LIN {X 0,Y 426.471,Z 695.747,A -85,B 0,C 180,E1 10312.845,E2 10312.845} C_VEL
LIN {X 0,Y 420.657,Z 731.018,A -85,B 0,C 180,E1 10315.887,E2 10315.887} C_VEL
LIN {X 0,Y 414.924,Z 763.236,A -85,B 0,C 180,E1 10319.677,E2 10319.677} C_VEL
LIN {X 0,Y 409.909,Z 791.343,A -85,B 0,C 180,E1 10324.089,E2 10324.089} C_VEL
LIN {X 0,Y 406.178,Z 814.952,A -85,B 0,C 180,E1 10329.05,E2 10329.05} C_VEL
LIN {X 0,Y 403.918,Z 833.153,A -85,B 0,C 180,E1 10334.286,E2 10334.286} C_VEL
LIN {X 0,Y 403.628,Z 836.352,A -85,B 0,C 180,E1 10335.425,E2 10335.425} C_VEL
LIN {X 0,Y 400.755,Z 840.636,A -85,B 0,C 180,E1 10337.153,E2 10337.153} C_VEL
LIN {X 0,Y 395.126,Z 845.824,A -85,B 0,C 180,E1 10339.793,E2 10339.793} C_VEL
LIN {X 0,Y 395.001,Z 846.38,A -85,B 0,C 180,E1 10340.101,E2 10340.101} C_VEL
LIN {X 0,Y 394.597,Z 853.166,A -85,B 0,C 180,E1 10345.615,E2 10345.615} C_VEL
LIN {X 0,Y 394.715,Z 854.908,A -85,B 0,C 180,E1 10350.002,E2 10350.002} C_VEL
LIN {X 0,Y 394.613,Z 853.222,A -85,B 0,C 180,E1 10354.388,E2 10354.388} C_VEL
LIN {X 0,Y 394.945,Z 846.511,A -85,B 0,C 180,E1 10359.902,E2 10359.902} C_VEL
LIN {X 0,Y 395.944,Z 834.241,A -85,B 0,C 180,E1 10365.475,E2 10365.475} C_VEL
LIN {X 0,Y 398.38,Z 815.704,A -85,B 0,C 180,E1 10371.093,E2 10371.093} C_VEL
LIN {X 0,Y 402.285,Z 792.827,A -85,B 0,C 180,E1 10376.109,E2 10376.109} C_VEL
LIN {X 0,Y 407.51,Z 765.346,A -85,B 0,C 180,E1 10380.61,E2 10380.61} C_VEL
LIN {X 0,Y 413.404,Z 734.349,A -85,B 0,C 180,E1 10384.414,E2 10384.414} C_VEL
LIN {X 0,Y 419.63,Z 699.188,A -85,B 0,C 180,E1 10387.577,E2 10387.577} C_VEL
LIN {X 0,Y 424.895,Z 663.712,A -85,B 0,C 180,E1 10389.841,E2 10389.841} C_VEL
LIN {X 0,Y 429.031,Z 626.267,A -85,B 0,C 180,E1 10391.417,E2 10391.417} C_VEL
LIN {X 0,Y 428.573,Z 619.383,A -85,B 0,C 180,E1 10391.743,E2 10391.743} C_VEL
LIN {X 0,Y 412.157,Z 584.483,A -85,B 0,C 180,E1 10394.597,E2 10394.597} C_VEL
LIN {X 0,Y 393.303,Z 551.113,A -85,B 0,C 180,E1 10397.831,E2 10397.831} C_VEL
LIN {X 0,Y 393.107,Z 549.53,A -85,B 0,C 180,E1 10397.988,E2 10397.988} C_VEL
LIN {X 0,Y 393.066,Z 549.53,A -85,B 0,C 180,E1 10404.827,E2 10404.827} C_VEL
LIN {X 0,Y 393.133,Z 549.53,A -85,B 0,C 180,E1 10411.99,E2 10411.99} C_VEL
LIN {X 0,Y 393.428,Z 549.53,A -85,B 0,C 180,E1 10417.432,E2 10417.432} C_VEL
LIN {X 0,Y 393.65,Z 549.53,A -85,B 0,C 180,E1 10424.419,E2 10424.419} C_VEL
LIN {X 0,Y 393.977,Z 549.53,A -85,B 0,C 180,E1 10431.171,E2 10431.171} C_VEL
LIN {X 0,Y 394.49,Z 549.53,A -85,B 0,C 180,E1 10437.79,E2 10437.79} C_VEL
LIN {X 0,Y 394.273,Z 549.53,A -85,B 0,C 180,E1 10444.371,E2 10444.371} C_VEL
LIN {X 0,Y 393.966,Z 549.53,A -85,B 0,C 180,E1 10451.02,E2 10451.02} C_VEL
LIN {X 0,Y 393.651,Z 549.53,A -85,B 0,C 180,E1 10457.835,E2 10457.835} C_VEL
LIN {X 0,Y 393.41,Z 549.53,A -85,B 0,C 180,E1 10464.93,E2 10464.93} C_VEL
LIN {X 0,Y 393.257,Z 549.53,A -85,B 0,C 180,E1 10472.464,E2 10472.464} C_VEL
LIN {X 0,Y 393.138,Z 549.53,A -85,B 0,C 180,E1 10479.852,E2 10479.852} C_VEL
LIN {X 0,Y 393.035,Z 549.53,A -85,B 0,C 180,E1 10486.802,E2 10486.802} C_VEL
LIN {X 0,Y 393.151,Z 549.53,A -85,B 0,C 180,E1 10493.661,E2 10493.661} C_VEL
LIN {X 0,Y 393.294,Z 549.53,A -85,B 0,C 180,E1 10500.078,E2 10500.078} C_VEL
LIN {X 0,Y 393.473,Z 549.53,A -85,B 0,C 180,E1 10507.447,E2 10507.447} C_VEL
LIN {X 0,Y 393.748,Z 549.858,A -85,B 0,C 180,E1 10514.366,E2 10514.366} C_VEL
LIN {X 0,Y 398.982,Z 560.257,A -85,B 0,C 180,E1 10515.316,E2 10515.316} C_VEL
LIN {X 0,Y 415.159,Z 593.265,A -85,B 0,C 180,E1 10518.486,E2 10518.486} C_VEL
LIN {X 0,Y 422.389,Z 615.31,A -85,B 0,C 180,E1 10520.492,E2 10520.492} C_VEL
LIN {X 0,Y 417.734,Z 650.048,A -85,B 0,C 180,E1 10522.702,E2 10522.702} C_VEL
LIN {X 0,Y 412.529,Z 681.161,A -85,B 0,C 180,E1 10525.54,E2 10525.54} C_VEL
LIN {X 0,Y 406.889,Z 710.862,A -85,B 0,C 180,E1 10529.292,E2 10529.292} C_VEL
LIN {X 0,Y 401.898,Z 736.31,A -85,B 0,C 180,E1 10533.766,E2 10533.766} C_VEL
LIN {X 0,Y 398.293,Z 756.361,A -85,B 0,C 180,E1 10538.715,E2 10538.715} C_VEL
LIN {X 0,Y 396.006,Z 771.387,A -85,B 0,C 180,E1 10544.145,E2 10544.145} C_VEL
LIN {X 0,Y 395.061,Z 779.568,A -85,B 0,C 180,E1 10548.944,E2 10548.944} C_VEL
LIN {X 0,Y 394.329,Z 783.387,A -85,B 0,C 180,E1 10553.38,E2 10553.38} C_VEL
LIN {X 0,Y 394.392,Z 783.535,A -85,B 0,C 180,E1 10558.419,E2 10558.419} C_VEL
LIN {X 0,Y 395.372,Z 778.667,A -85,B 0,C 180,E1 10563.847,E2 10563.847} C_VEL
LIN {X 0,Y 396.658,Z 768.466,A -85,B 0,C 180,E1 10569.268,E2 10569.268} C_VEL
LIN {X 0,Y 399.169,Z 752.985,A -85,B 0,C 180,E1 10574.422,E2 10574.422} C_VEL
LIN {X 0,Y 403.09,Z 732.77,A -85,B 0,C 180,E1 10579.115,E2 10579.115} C_VEL
LIN {X 0,Y 408.186,Z 708.039,A -85,B 0,C 180,E1 10583.279,E2 10583.279} C_VEL
LIN {X 0,Y 413.987,Z 678.023,A -85,B 0,C 180,E1 10586.965,E2 10586.965} C_VEL
LIN {X 0,Y 419.505,Z 645.504,A -85,B 0,C 180,E1 10589.789,E2 10589.789} C_VEL
LIN {X 0,Y 423.419,Z 614.726,A -85,B 0,C 180,E1 10591.704,E2 10591.704} C_VEL
LIN {X 0,Y 410.683,Z 582.196,A -85,B 0,C 180,E1 10594.957,E2 10594.957} C_VEL
LIN {X 0,Y 395.046,Z 554.114,A -85,B 0,C 180,E1 10598.086,E2 10598.086} C_VEL
LIN {X 0,Y 393.557,Z 549.53,A -85,B 0,C 180,E1 10598.516,E2 10598.516} C_VEL
LIN {X 0,Y 393.66,Z 549.53,A -85,B 0,C 180,E1 10604.458,E2 10604.458} C_VEL
LIN {X 0,Y 393.997,Z 549.53,A -85,B 0,C 180,E1 10611.208,E2 10611.208} C_VEL
LIN {X 0,Y 394.47,Z 549.53,A -85,B 0,C 180,E1 10617.826,E2 10617.826} C_VEL
LIN {X 0,Y 394.267,Z 549.53,A -85,B 0,C 180,E1 10624.407,E2 10624.407} C_VEL
LIN {X 0,Y 393.97,Z 549.53,A -85,B 0,C 180,E1 10631.057,E2 10631.057} C_VEL
LIN {X 0,Y 393.667,Z 549.53,A -85,B 0,C 180,E1 10637.873,E2 10637.873} C_VEL
LIN {X 0,Y 393.385,Z 549.53,A -85,B 0,C 180,E1 10644.972,E2 10644.972} C_VEL
LIN {X 0,Y 393.268,Z 549.53,A -85,B 0,C 180,E1 10652.506,E2 10652.506} C_VEL
LIN {X 0,Y 393.117,Z 549.53,A -85,B 0,C 180,E1 10659.853,E2 10659.853} C_VEL
LIN {X 0,Y 393.019,Z 549.552,A -85,B 0,C 180,E1 10661.786,E2 10661.786} C_VEL
LIN {X 0,Y 395.349,Z 555.078,A -85,B 0,C 180,E1 10662.289,E2 10662.289} C_VEL
LIN {X 0,Y 414.303,Z 587.868,A -85,B 0,C 180,E1 10665.71,E2 10665.71} C_VEL
LIN {X 0,Y 429.06,Z 620.928,A -85,B 0,C 180,E1 10668.451,E2 10668.451} C_VEL
LIN {X 0,Y 424.831,Z 660.824,A -85,B 0,C 180,E1 10670.072,E2 10670.072} C_VEL
LIN {X 0,Y 419.322,Z 698.722,A -85,B 0,C 180,E1 10672.477,E2 10672.477} C_VEL
LIN {X 0,Y 413.275,Z 733.396,A -85,B 0,C 180,E1 10675.601,E2 10675.601} C_VEL
LIN {X 0,Y 407.388,Z 764.437,A -85,B 0,C 180,E1 10679.384,E2 10679.384} C_VEL
LIN {X 0,Y 402.203,Z 792.195,A -85,B 0,C 180,E1 10683.894,E2 10683.894} C_VEL
LIN {X 0,Y 398.349,Z 815.265,A -85,B 0,C 180,E1 10688.909,E2 10688.909} C_VEL
LIN {X 0,Y 395.954,Z 833.988,A -85,B 0,C 180,E1 10694.529,E2 10694.529} C_VEL
LIN {X 0,Y 395.001,Z 846.38,A -85,B 0,C 180,E1 10700.101,E2 10700.101} C_VEL
LIN {X 0,Y 392.28,Z 849.129,A -85,B 0,C 180,E1 10701.929,E2 10701.929} C_VEL
LIN {X 0,Y 386.796,Z 851.796,A -85,B 0,C 180,E1 10704.721,E2 10704.721} C_VEL
LIN {X 0,Y 386.707,Z 852.052,A -85,B 0,C 180,E1 10705.046,E2 10705.046} C_VEL
LIN {X 0,Y 386.852,Z 854.204,A -85,B 0,C 180,E1 10710.002,E2 10710.002} C_VEL
LIN {X 0,Y 386.746,Z 852.519,A -85,B 0,C 180,E1 10714.477,E2 10714.477} C_VEL
LIN {X 0,Y 387.089,Z 845.8,A -85,B 0,C 180,E1 10720.105,E2 10720.105} C_VEL
LIN {X 0,Y 388.13,Z 833.511,A -85,B 0,C 180,E1 10725.794,E2 10725.794} C_VEL
LIN {X 0,Y 390.582,Z 815.874,A -85,B 0,C 180,E1 10731.288,E2 10731.288} C_VEL
LIN {X 0,Y 394.703,Z 793.039,A -85,B 0,C 180,E1 10736.444,E2 10736.444} C_VEL
LIN {X 0,Y 400.02,Z 766.445,A -85,B 0,C 180,E1 10740.931,E2 10740.931} C_VEL
LIN {X 0,Y 406.373,Z 734.587,A -85,B 0,C 180,E1 10744.942,E2 10744.942} C_VEL
LIN {X 0,Y 412.893,Z 699.726,A -85,B 0,C 180,E1 10748.14,E2 10748.14} C_VEL
LIN {X 0,Y 418.485,Z 663.769,A -85,B 0,C 180,E1 10750.473,E2 10750.473} C_VEL
LIN {X 0,Y 422.776,Z 626.655,A -85,B 0,C 180,E1 10752.06,E2 10752.06} C_VEL
LIN {X 0,Y 421.658,Z 620.596,A -85,B 0,C 180,E1 10752.433,E2 10752.433} C_VEL
LIN {X 0,Y 405.945,Z 587.248,A -85,B 0,C 180,E1 10755.297,E2 10755.297} C_VEL
LIN {X 0,Y 386.357,Z 553.583,A -85,B 0,C 180,E1 10758.759,E2 10758.759} C_VEL
LIN {X 0,Y 385.217,Z 549.53,A -85,B 0,C 180,E1 10759.111,E2 10759.111} C_VEL
LIN {X 0,Y 385.118,Z 549.53,A -85,B 0,C 180,E1 10766.718,E2 10766.718} C_VEL
LIN {X 0,Y 385.314,Z 549.53,A -85,B 0,C 180,E1 10774.261,E2 10774.261} C_VEL
LIN {X 0,Y 385.665,Z 549.53,A -85,B 0,C 180,E1 10779.899,E2 10779.899} C_VEL
LIN {X 0,Y 385.782,Z 549.53,A -85,B 0,C 180,E1 10786.41,E2 10786.41} C_VEL
LIN {X 0,Y 386.241,Z 549.53,A -85,B 0,C 180,E1 10793.252,E2 10793.252} C_VEL
LIN {X 0,Y 386.542,Z 549.53,A -85,B 0,C 180,E1 10799.981,E2 10799.981} C_VEL
LIN {X 0,Y 386.242,Z 549.53,A -85,B 0,C 180,E1 10806.711,E2 10806.711} C_VEL
LIN {X 0,Y 385.971,Z 549.53,A -85,B 0,C 180,E1 10813.544,E2 10813.544} C_VEL
LIN {X 0,Y 385.622,Z 549.53,A -85,B 0,C 180,E1 10820.596,E2 10820.596} C_VEL
LIN {X 0,Y 385.391,Z 549.53,A -85,B 0,C 180,E1 10827.997,E2 10827.997} C_VEL
LIN {X 0,Y 385.257,Z 549.53,A -85,B 0,C 180,E1 10835.949,E2 10835.949} C_VEL
LIN {X 0,Y 385.08,Z 549.53,A -85,B 0,C 180,E1 10841.877,E2 10841.877} C_VEL
LIN {X 0,Y 385.068,Z 549.53,A -85,B 0,C 180,E1 10848.223,E2 10848.223} C_VEL
LIN {X 0,Y 385.242,Z 549.53,A -85,B 0,C 180,E1 10854.014,E2 10854.014} C_VEL
LIN {X 0,Y 385.337,Z 549.53,A -85,B 0,C 180,E1 10859.43,E2 10859.43} C_VEL
LIN {X 0,Y 385.58,Z 549.53,A -85,B 0,C 180,E1 10866.959,E2 10866.959} C_VEL
LIN {X 0,Y 385.772,Z 549.53,A -85,B 0,C 180,E1 10873.251,E2 10873.251} C_VEL
LIN {X 0,Y 388.253,Z 555.254,A -85,B 0,C 180,E1 10873.76,E2 10873.76} C_VEL
LIN {X 0,Y 405.744,Z 588.831,A -85,B 0,C 180,E1 10877.194,E2 10877.194} C_VEL
LIN {X 0,Y 415.978,Z 616.303,A -85,B 0,C 180,E1 10879.879,E2 10879.879} C_VEL
LIN {X 0,Y 411.293,Z 649.927,A -85,B 0,C 180,E1 10882.038,E2 10882.038} C_VEL
LIN {X 0,Y 405.76,Z 681.449,A -85,B 0,C 180,E1 10884.931,E2 10884.931} C_VEL
LIN {X 0,Y 400.146,Z 709.999,A -85,B 0,C 180,E1 10888.562,E2 10888.562} C_VEL
LIN {X 0,Y 394.861,Z 735.482,A -85,B 0,C 180,E1 10893.01,E2 10893.01} C_VEL
LIN {X 0,Y 391.051,Z 754.99,A -85,B 0,C 180,E1 10897.76,E2 10897.76} C_VEL
LIN {X 0,Y 388.554,Z 769.773,A -85,B 0,C 180,E1 10902.902,E2 10902.902} C_VEL
LIN {X 0,Y 387.354,Z 779.383,A -85,B 0,C 180,E1 10908.157,E2 10908.157} C_VEL
LIN {X 0,Y 386.51,Z 783.925,A -85,B 0,C 180,E1 10912.979,E2 10912.979} C_VEL
LIN {X 0,Y 386.471,Z 784.476,A -85,B 0,C 180,E1 10917.938,E2 10917.938} C_VEL
LIN {X 0,Y 387.377,Z 780.657,A -85,B 0,C 180,E1 10923.048,E2 10923.048} C_VEL
LIN {X 0,Y 388.494,Z 771.732,A -85,B 0,C 180,E1 10928.422,E2 10928.422} C_VEL
LIN {X 0,Y 390.929,Z 757.617,A -85,B 0,C 180,E1 10933.652,E2 10933.652} C_VEL
LIN {X 0,Y 394.939,Z 737.673,A -85,B 0,C 180,E1 10938.728,E2 10938.728} C_VEL
LIN {X 0,Y 400.489,Z 712.216,A -85,B 0,C 180,E1 10943.311,E2 10943.311} C_VEL
LIN {X 0,Y 406.474,Z 683.127,A -85,B 0,C 180,E1 10947.082,E2 10947.082} C_VEL
LIN {X 0,Y 412.498,Z 650.226,A -85,B 0,C 180,E1 10950.129,E2 10950.129} C_VEL
LIN {X 0,Y 416.669,Z 616.289,A -85,B 0,C 180,E1 10952.38,E2 10952.38} C_VEL
LIN {X 0,Y 403.829,Z 583.58,A -85,B 0,C 180,E1 10955.816,E2 10955.816} C_VEL
LIN {X 0,Y 388.017,Z 555.131,A -85,B 0,C 180,E1 10959.166,E2 10959.166} C_VEL
LIN {X 0,Y 385.726,Z 549.53,A -85,B 0,C 180,E1 10959.865,E2 10959.865} C_VEL
LIN {X 0,Y 385.803,Z 549.53,A -85,B 0,C 180,E1 10966.45,E2 10966.45} C_VEL
LIN {X 0,Y 386.278,Z 549.53,A -85,B 0,C 180,E1 10973.29,E2 10973.29} C_VEL
LIN {X 0,Y 386.548,Z 549.53,A -85,B 0,C 180,E1 10980.019,E2 10980.019} C_VEL
LIN {X 0,Y 386.244,Z 549.53,A -85,B 0,C 180,E1 10986.748,E2 10986.748} C_VEL
LIN {X 0,Y 385.991,Z 549.53,A -85,B 0,C 180,E1 10993.582,E2 10993.582} C_VEL
LIN {X 0,Y 385.615,Z 549.53,A -85,B 0,C 180,E1 11000.636,E2 11000.636} C_VEL
LIN {X 0,Y 385.387,Z 549.53,A -85,B 0,C 180,E1 11008.04,E2 11008.04} C_VEL
LIN {X 0,Y 385.233,Z 549.53,A -85,B 0,C 180,E1 11014.657,E2 11014.657} C_VEL
LIN {X 0,Y 385.198,Z 549.884,A -85,B 0,C 180,E1 11020.518,E2 11020.518} C_VEL
LIN {X 0,Y 387.642,Z 555.268,A -85,B 0,C 180,E1 11021.073,E2 11021.073} C_VEL
LIN {X 0,Y 406.583,Z 587.415,A -85,B 0,C 180,E1 11024.695,E2 11024.695} C_VEL
LIN {X 0,Y 421.438,Z 620.064,A -85,B 0,C 180,E1 11027.575,E2 11027.575} C_VEL
LIN {X 0,Y 422.509,Z 626.284,A -85,B 0,C 180,E1 11027.955,E2 11027.955} C_VEL
LIN {X 0,Y 417.796,Z 666.137,A -85,B 0,C 180,E1 11029.705,E2 11029.705} C_VEL
LIN {X 0,Y 411.485,Z 705.521,A -85,B 0,C 180,E1 11032.405,E2 11032.405} C_VEL
LIN {X 0,Y 404.886,Z 740.387,A -85,B 0,C 180,E1 11035.816,E2 11035.816} C_VEL
LIN {X 0,Y 398.767,Z 771.137,A -85,B 0,C 180,E1 11039.909,E2 11039.909} C_VEL
LIN {X 0,Y 393.725,Z 797.105,A -85,B 0,C 180,E1 11044.51,E2 11044.51} C_VEL
LIN {X 0,Y 389.994,Z 819.77,A -85,B 0,C 180,E1 11049.917,E2 11049.917} C_VEL
LIN {X 0,Y 387.878,Z 836.124,A -85,B 0,C 180,E1 11055.354,E2 11055.354} C_VEL
LIN {X 0,Y 386.98,Z 847.395,A -85,B 0,C 180,E1 11061.028,E2 11061.028} C_VEL
LIN {X 0,Y 386.707,Z 852.052,A -85,B 0,C 180,E1 11065.046,E2 11065.046} C_VEL
LIN {X 0,Y 384.331,Z 853.217,A -85,B 0,C 180,E1 11066.952,E2 11066.952} C_VEL
LIN {X 0,Y 378.98,Z 853.469,A -85,B 0,C 180,E1 11070.169,E2 11070.169} C_VEL
LIN {X 0,Y 378.856,Z 851.309,A -85,B 0,C 180,E1 11075.212,E2 11075.212} C_VEL
LIN {X 0,Y 379.22,Z 845.088,A -85,B 0,C 180,E1 11080.317,E2 11080.317} C_VEL
LIN {X 0,Y 380.334,Z 832.776,A -85,B 0,C 180,E1 11086.127,E2 11086.127} C_VEL
LIN {X 0,Y 382.893,Z 815.414,A -85,B 0,C 180,E1 11091.654,E2 11091.654} C_VEL
LIN {X 0,Y 387.461,Z 791.705,A -85,B 0,C 180,E1 11097.086,E2 11097.086} C_VEL
LIN {X 0,Y 393.329,Z 763.563,A -85,B 0,C 180,E1 11101.84,E2 11101.84} C_VEL
LIN {X 0,Y 399.84,Z 732.637,A -85,B 0,C 180,E1 11105.722,E2 11105.722} C_VEL
LIN {X 0,Y 406.572,Z 698.065,A -85,B 0,C 180,E1 11108.888,E2 11108.888} C_VEL
LIN {X 0,Y 412.308,Z 662.252,A -85,B 0,C 180,E1 11111.209,E2 11111.209} C_VEL
LIN {X 0,Y 416.143,Z 625.507,A -85,B 0,C 180,E1 11112.836,E2 11112.836} C_VEL
LIN {X 0,Y 400.463,Z 591.124,A -85,B 0,C 180,E1 11115.903,E2 11115.903} C_VEL
LIN {X 0,Y 379.231,Z 554.747,A -85,B 0,C 180,E1 11119.79,E2 11119.79} C_VEL
LIN {X 0,Y 377.267,Z 549.53,A -85,B 0,C 180,E1 11120.323,E2 11120.323} C_VEL
LIN {X 0,Y 377.174,Z 549.53,A -85,B 0,C 180,E1 11127.162,E2 11127.162} C_VEL
LIN {X 0,Y 377.369,Z 549.53,A -85,B 0,C 180,E1 11133.89,E2 11133.89} C_VEL
LIN {X 0,Y 377.629,Z 549.53,A -85,B 0,C 180,E1 11138.907,E2 11138.907} C_VEL
LIN {X 0,Y 377.84,Z 549.53,A -85,B 0,C 180,E1 11146.119,E2 11146.119} C_VEL
LIN {X 0,Y 378.321,Z 549.53,A -85,B 0,C 180,E1 11153.11,E2 11153.11} C_VEL
LIN {X 0,Y 378.64,Z 549.53,A -85,B 0,C 180,E1 11159.981,E2 11159.981} C_VEL
LIN {X 0,Y 378.323,Z 549.53,A -85,B 0,C 180,E1 11166.852,E2 11166.852} C_VEL
LIN {X 0,Y 378.018,Z 549.53,A -85,B 0,C 180,E1 11173.835,E2 11173.835} C_VEL
LIN {X 0,Y 377.654,Z 549.53,A -85,B 0,C 180,E1 11181.051,E2 11181.051} C_VEL
LIN {X 0,Y 377.412,Z 549.53,A -85,B 0,C 180,E1 11188.643,E2 11188.643} C_VEL
LIN {X 0,Y 377.316,Z 549.53,A -85,B 0,C 180,E1 11194.017,E2 11194.017} C_VEL
LIN {X 0,Y 377.128,Z 549.53,A -85,B 0,C 180,E1 11200.511,E2 11200.511} C_VEL
LIN {X 0,Y 377.055,Z 549.53,A -85,B 0,C 180,E1 11207.126,E2 11207.126} C_VEL
LIN {X 0,Y 377.278,Z 549.53,A -85,B 0,C 180,E1 11213.131,E2 11213.131} C_VEL
LIN {X 0,Y 377.315,Z 549.53,A -85,B 0,C 180,E1 11218.671,E2 11218.671} C_VEL
LIN {X 0,Y 377.485,Z 549.53,A -85,B 0,C 180,E1 11223.911,E2 11223.911} C_VEL
LIN {X 0,Y 377.655,Z 549.53,A -85,B 0,C 180,E1 11228.921,E2 11228.921} C_VEL
LIN {X 0,Y 377.839,Z 550.299,A -85,B 0,C 180,E1 11232.134,E2 11232.134} C_VEL
LIN {X 0,Y 386.756,Z 566.255,A -85,B 0,C 180,E1 11233.872,E2 11233.872} C_VEL
LIN {X 0,Y 402.213,Z 598.37,A -85,B 0,C 180,E1 11237.249,E2 11237.249} C_VEL
LIN {X 0,Y 409.274,Z 619.687,A -85,B 0,C 180,E1 11239.375,E2 11239.375} C_VEL
LIN {X 0,Y 404.372,Z 652.868,A -85,B 0,C 180,E1 11241.596,E2 11241.596} C_VEL
LIN {X 0,Y 398.419,Z 685.269,A -85,B 0,C 180,E1 11244.701,E2 11244.701} C_VEL
LIN {X 0,Y 392.241,Z 714.458,A -85,B 0,C 180,E1 11248.61,E2 11248.61} C_VEL
LIN {X 0,Y 387.03,Z 738.331,A -85,B 0,C 180,E1 11253.032,E2 11253.032} C_VEL
LIN {X 0,Y 383.147,Z 757.412,A -85,B 0,C 180,E1 11257.922,E2 11257.922} C_VEL
LIN {X 0,Y 380.662,Z 771.669,A -85,B 0,C 180,E1 11263.174,E2 11263.174} C_VEL
LIN {X 0,Y 379.412,Z 780.815,A -85,B 0,C 180,E1 11268.551,E2 11268.551} C_VEL
LIN {X 0,Y 378.56,Z 784.947,A -85,B 0,C 180,E1 11273.612,E2 11273.612} C_VEL
LIN {X 0,Y 378.668,Z 784.848,A -85,B 0,C 180,E1 11278.816,E2 11278.816} C_VEL
LIN {X 0,Y 379.698,Z 780.606,A -85,B 0,C 180,E1 11283.805,E2 11283.805} C_VEL
LIN {X 0,Y 381.021,Z 771.083,A -85,B 0,C 180,E1 11289.319,E2 11289.319} C_VEL
LIN {X 0,Y 383.821,Z 756.168,A -85,B 0,C 180,E1 11294.707,E2 11294.707} C_VEL
LIN {X 0,Y 388.411,Z 735.173,A -85,B 0,C 180,E1 11299.888,E2 11299.888} C_VEL
LIN {X 0,Y 394.245,Z 709.826,A -85,B 0,C 180,E1 11304.335,E2 11304.335} C_VEL
LIN {X 0,Y 400.47,Z 680.842,A -85,B 0,C 180,E1 11308.032,E2 11308.032} C_VEL
LIN {X 0,Y 406.786,Z 647.048,A -85,B 0,C 180,E1 11311.08,E2 11311.08} C_VEL
LIN {X 0,Y 410.49,Z 619.762,A -85,B 0,C 180,E1 11312.878,E2 11312.878} C_VEL
LIN {X 0,Y 398.576,Z 588.31,A -85,B 0,C 180,E1 11316.32,E2 11316.32} C_VEL
LIN {X 0,Y 383.84,Z 561.006,A -85,B 0,C 180,E1 11319.68,E2 11319.68} C_VEL
LIN {X 0,Y 377.85,Z 550.7,A -85,B 0,C 180,E1 11321.051,E2 11321.051} C_VEL
LIN {X 0,Y 377.75,Z 549.53,A -85,B 0,C 180,E1 11321.387,E2 11321.387} C_VEL
LIN {X 0,Y 377.972,Z 549.53,A -85,B 0,C 180,E1 11328.507,E2 11328.507} C_VEL
LIN {X 0,Y 378.437,Z 549.53,A -85,B 0,C 180,E1 11335.446,E2 11335.446} C_VEL
LIN {X 0,Y 378.522,Z 549.53,A -85,B 0,C 180,E1 11342.303,E2 11342.303} C_VEL
LIN {X 0,Y 378.167,Z 549.53,A -85,B 0,C 180,E1 11349.202,E2 11349.202} C_VEL
LIN {X 0,Y 377.888,Z 549.53,A -85,B 0,C 180,E1 11356.248,E2 11356.248} C_VEL
LIN {X 0,Y 377.554,Z 549.53,A -85,B 0,C 180,E1 11363.573,E2 11363.573} C_VEL
LIN {X 0,Y 377.416,Z 549.53,A -85,B 0,C 180,E1 11368.686,E2 11368.686} C_VEL
LIN {X 0,Y 377.316,Z 549.53,A -85,B 0,C 180,E1 11374.063,E2 11374.063} C_VEL
LIN {X 0,Y 377.31,Z 549.53,A -85,B 0,C 180,E1 11379.073,E2 11379.073} C_VEL
LIN {X 0,Y 379.801,Z 555.282,A -85,B 0,C 180,E1 11379.732,E2 11379.732} C_VEL
LIN {X 0,Y 398.809,Z 586.851,A -85,B 0,C 180,E1 11383.605,E2 11383.605} C_VEL
LIN {X 0,Y 413.991,Z 619.607,A -85,B 0,C 180,E1 11386.687,E2 11386.687} C_VEL
LIN {X 0,Y 416.364,Z 626.906,A -85,B 0,C 180,E1 11387.283,E2 11387.283} C_VEL
LIN {X 0,Y 411.311,Z 667.365,A -85,B 0,C 180,E1 11389.109,E2 11389.109} C_VEL
LIN {X 0,Y 404.88,Z 705.412,A -85,B 0,C 180,E1 11391.777,E2 11391.777} C_VEL
LIN {X 0,Y 398.055,Z 739.668,A -85,B 0,C 180,E1 11395.175,E2 11395.175} C_VEL
LIN {X 0,Y 391.625,Z 770.248,A -85,B 0,C 180,E1 11399.301,E2 11399.301} C_VEL
LIN {X 0,Y 386.151,Z 796.925,A -85,B 0,C 180,E1 11404.12,E2 11404.12} C_VEL
LIN {X 0,Y 382.272,Z 818.957,A -85,B 0,C 180,E1 11409.494,E2 11409.494} C_VEL
LIN {X 0,Y 380.047,Z 835.356,A -85,B 0,C 180,E1 11415.045,E2 11415.045} C_VEL
LIN {X 0,Y 379.112,Z 846.657,A -85,B 0,C 180,E1 11420.84,E2 11420.84} C_VEL
LIN {X 0,Y 378.849,Z 851.732,A -85,B 0,C 180,E1 11425.433,E2 11425.433} C_VEL
LIN {X 0,Y 378.98,Z 853.469,A -85,B 0,C 180,E1 11430.169,E2 11430.169} C_VEL
LIN {X 0,Y 376.344,Z 852.926,A -85,B 0,C 180,E1 11432.113,E2 11432.113} C_VEL
LIN {X 0,Y 370.977,Z 850.565,A -85,B 0,C 180,E1 11435.366,E2 11435.366} C_VEL
LIN {X 0,Y 371.342,Z 844.372,A -85,B 0,C 180,E1 11440.538,E2 11440.538} C_VEL
LIN {X 0,Y 372.556,Z 832.039,A -85,B 0,C 180,E1 11446.473,E2 11446.473} C_VEL
LIN {X 0,Y 375.503,Z 813.491,A -85,B 0,C 180,E1 11452.421,E2 11452.421} C_VEL
LIN {X 0,Y 380.244,Z 790.146,A -85,B 0,C 180,E1 11457.797,E2 11457.797} C_VEL
LIN {X 0,Y 386.345,Z 762.665,A -85,B 0,C 180,E1 11462.485,E2 11462.485} C_VEL
LIN {X 0,Y 393.184,Z 731.684,A -85,B 0,C 180,E1 11466.41,E2 11466.41} C_VEL
LIN {X 0,Y 400.235,Z 696.848,A -85,B 0,C 180,E1 11469.623,E2 11469.623} C_VEL
LIN {X 0,Y 406.363,Z 659.625,A -85,B 0,C 180,E1 11472.027,E2 11472.027} C_VEL
LIN {X 0,Y 409.851,Z 628.218,A -85,B 0,C 180,E1 11473.435,E2 11473.435} C_VEL
LIN {X 0,Y 394.517,Z 594.497,A -85,B 0,C 180,E1 11476.582,E2 11476.582} C_VEL
LIN {X 0,Y 374.605,Z 560.065,A -85,B 0,C 180,E1 11480.365,E2 11480.365} C_VEL
LIN {X 0,Y 369.429,Z 550.458,A -85,B 0,C 180,E1 11481.459,E2 11481.459} C_VEL
LIN {X 0,Y 369.384,Z 549.53,A -85,B 0,C 180,E1 11481.602,E2 11481.602} C_VEL
LIN {X 0,Y 369.249,Z 549.53,A -85,B 0,C 180,E1 11489.119,E2 11489.119} C_VEL
LIN {X 0,Y 369.527,Z 549.53,A -85,B 0,C 180,E1 11495.883,E2 11495.883} C_VEL
LIN {X 0,Y 369.849,Z 549.53,A -85,B 0,C 180,E1 11503.389,E2 11503.389} C_VEL
LIN {X 0,Y 370.162,Z 549.53,A -85,B 0,C 180,E1 11510.598,E2 11510.598} C_VEL
LIN {X 0,Y 370.762,Z 549.53,A -85,B 0,C 180,E1 11517.649,E2 11517.649} C_VEL
LIN {X 0,Y 370.539,Z 549.53,A -85,B 0,C 180,E1 11524.651,E2 11524.651} C_VEL
LIN {X 0,Y 370.163,Z 549.53,A -85,B 0,C 180,E1 11531.925,E2 11531.925} C_VEL
LIN {X 0,Y 369.799,Z 549.53,A -85,B 0,C 180,E1 11539.028,E2 11539.028} C_VEL
LIN {X 0,Y 369.499,Z 549.53,A -85,B 0,C 180,E1 11546.666,E2 11546.666} C_VEL
LIN {X 0,Y 369.425,Z 549.53,A -85,B 0,C 180,E1 11552.043,E2 11552.043} C_VEL
LIN {X 0,Y 369.227,Z 549.53,A -85,B 0,C 180,E1 11559.054,E2 11559.054} C_VEL
LIN {X 0,Y 369.141,Z 549.53,A -85,B 0,C 180,E1 11565.975,E2 11565.975} C_VEL
LIN {X 0,Y 369.254,Z 549.53,A -85,B 0,C 180,E1 11572.191,E2 11572.191} C_VEL
LIN {X 0,Y 369.397,Z 549.53,A -85,B 0,C 180,E1 11579.017,E2 11579.017} C_VEL
LIN {X 0,Y 369.611,Z 549.53,A -85,B 0,C 180,E1 11585.902,E2 11585.902} C_VEL
LIN {X 0,Y 369.773,Z 549.53,A -85,B 0,C 180,E1 11590.869,E2 11590.869} C_VEL
LIN {X 0,Y 372.261,Z 555.188,A -85,B 0,C 180,E1 11591.425,E2 11591.425} C_VEL
LIN {X 0,Y 389.181,Z 585.887,A -85,B 0,C 180,E1 11594.967,E2 11594.967} C_VEL
LIN {X 0,Y 401.619,Z 617.364,A -85,B 0,C 180,E1 11598.334,E2 11598.334} C_VEL
LIN {X 0,Y 402.526,Z 623.665,A -85,B 0,C 180,E1 11598.89,E2 11598.89} C_VEL
LIN {X 0,Y 397.073,Z 658.603,A -85,B 0,C 180,E1 11601.378,E2 11601.378} C_VEL
LIN {X 0,Y 390.749,Z 690.115,A -85,B 0,C 180,E1 11604.597,E2 11604.597} C_VEL
LIN {X 0,Y 384.479,Z 718.191,A -85,B 0,C 180,E1 11608.582,E2 11608.582} C_VEL
LIN {X 0,Y 379.018,Z 742.125,A -85,B 0,C 180,E1 11613.269,E2 11613.269} C_VEL
LIN {X 0,Y 374.902,Z 761.591,A -85,B 0,C 180,E1 11618.68,E2 11618.68} C_VEL
LIN {X 0,Y 372.55,Z 774.694,A -85,B 0,C 180,E1 11624.064,E2 11624.064} C_VEL
LIN {X 0,Y 371.477,Z 782.169,A -85,B 0,C 180,E1 11628.962,E2 11628.962} C_VEL
LIN {X 0,Y 370.669,Z 785.856,A -85,B 0,C 180,E1 11634.021,E2 11634.021} C_VEL
LIN {X 0,Y 370.854,Z 785.429,A -85,B 0,C 180,E1 11639.226,E2 11639.226} C_VEL
LIN {X 0,Y 371.97,Z 780.558,A -85,B 0,C 180,E1 11644.606,E2 11644.606} C_VEL
LIN {X 0,Y 373.613,Z 770.429,A -85,B 0,C 180,E1 11650.256,E2 11650.256} C_VEL
LIN {X 0,Y 376.8,Z 754.686,A -85,B 0,C 180,E1 11655.769,E2 11655.769} C_VEL
LIN {X 0,Y 381.638,Z 734.007,A -85,B 0,C 180,E1 11660.79,E2 11660.79} C_VEL
LIN {X 0,Y 388.097,Z 707.581,A -85,B 0,C 180,E1 11665.375,E2 11665.375} C_VEL
LIN {X 0,Y 394.752,Z 677.462,A -85,B 0,C 180,E1 11669.112,E2 11669.112} C_VEL
LIN {X 0,Y 401.015,Z 644.752,A -85,B 0,C 180,E1 11671.99,E2 11671.99} C_VEL
LIN {X 0,Y 404.259,Z 623.006,A -85,B 0,C 180,E1 11673.415,E2 11673.415} C_VEL
LIN {X 0,Y 393.005,Z 592.131,A -85,B 0,C 180,E1 11676.938,E2 11676.938} C_VEL
LIN {X 0,Y 377.091,Z 562.149,A -85,B 0,C 180,E1 11680.823,E2 11680.823} C_VEL
LIN {X 0,Y 369.922,Z 550.971,A -85,B 0,C 180,E1 11682.55,E2 11682.55} C_VEL
LIN {X 0,Y 369.806,Z 549.53,A -85,B 0,C 180,E1 11682.658,E2 11682.658} C_VEL
LIN {X 0,Y 370.046,Z 549.53,A -85,B 0,C 180,E1 11688.258,E2 11688.258} C_VEL
LIN {X 0,Y 370.52,Z 549.53,A -85,B 0,C 180,E1 11695.348,E2 11695.348} C_VEL
LIN {X 0,Y 370.768,Z 549.53,A -85,B 0,C 180,E1 11700.019,E2 11700.019} C_VEL
LIN {X 0,Y 370.393,Z 549.53,A -85,B 0,C 180,E1 11707.038,E2 11707.038} C_VEL
LIN {X 0,Y 370.111,Z 549.53,A -85,B 0,C 180,E1 11714.177,E2 11714.177} C_VEL
LIN {X 0,Y 369.707,Z 549.53,A -85,B 0,C 180,E1 11721.568,E2 11721.568} C_VEL
LIN {X 0,Y 369.507,Z 549.53,A -85,B 0,C 180,E1 11726.709,E2 11726.709} C_VEL
LIN {X 0,Y 369.418,Z 549.53,A -85,B 0,C 180,E1 11732.089,E2 11732.089} C_VEL
LIN {X 0,Y 369.369,Z 549.53,A -85,B 0,C 180,E1 11737.549,E2 11737.549} C_VEL
LIN {X 0,Y 371.871,Z 555.241,A -85,B 0,C 180,E1 11738.257,E2 11738.257} C_VEL
LIN {X 0,Y 389.479,Z 583.535,A -85,B 0,C 180,E1 11742.124,E2 11742.124} C_VEL
LIN {X 0,Y 405.518,Z 616.29,A -85,B 0,C 180,E1 11745.489,E2 11745.489} C_VEL
LIN {X 0,Y 410.055,Z 630.165,A -85,B 0,C 180,E1 11746.69,E2 11746.69} C_VEL
LIN {X 0,Y 404.68,Z 669.57,A -85,B 0,C 180,E1 11748.559,E2 11748.559} C_VEL
LIN {X 0,Y 398.118,Z 706.304,A -85,B 0,C 180,E1 11751.212,E2 11751.212} C_VEL
LIN {X 0,Y 391.041,Z 739.988,A -85,B 0,C 180,E1 11754.633,E2 11754.633} C_VEL
LIN {X 0,Y 384.49,Z 769.382,A -85,B 0,C 180,E1 11758.668,E2 11758.668} C_VEL
LIN {X 0,Y 378.648,Z 796.663,A -85,B 0,C 180,E1 11763.699,E2 11763.699} C_VEL
LIN {X 0,Y 374.563,Z 818.155,A -85,B 0,C 180,E1 11769.052,E2 11769.052} C_VEL
LIN {X 0,Y 372.219,Z 834.587,A -85,B 0,C 180,E1 11774.723,E2 11774.723} C_VEL
LIN {X 0,Y 371.409,Z 844.154,A -85,B 0,C 180,E1 11779.467,E2 11779.467} C_VEL
LIN {X 0,Y 370.984,Z 851.015,A -85,B 0,C 180,E1 11785.335,E2 11785.335} C_VEL
LIN {X 0,Y 371.128,Z 852.772,A -85,B 0,C 180,E1 11790.138,E2 11790.138} C_VEL
LIN {X 0,Y 370.977,Z 850.565,A -85,B 0,C 180,E1 11795.366,E2 11795.366} C_VEL
LIN {X 0,Y 368.491,Z 848.539,A -85,B 0,C 180,E1 11797.337,E2 11797.337} C_VEL
LIN {X 0,Y 363.493,Z 844.425,A -85,B 0,C 180,E1 11800.285,E2 11800.285} C_VEL
LIN {X 0,Y 363.46,Z 843.866,A -85,B 0,C 180,E1 11800.624,E2 11800.624} C_VEL
LIN {X 0,Y 364.805,Z 831.303,A -85,B 0,C 180,E1 11806.833,E2 11806.833} C_VEL
LIN {X 0,Y 367.917,Z 812.7,A -85,B 0,C 180,E1 11812.91,E2 11812.91} C_VEL
LIN {X 0,Y 372.918,Z 789.304,A -85,B 0,C 180,E1 11818.392,E2 11818.392} C_VEL
LIN {X 0,Y 379.566,Z 760.939,A -85,B 0,C 180,E1 11823.274,E2 11823.274} C_VEL
LIN {X 0,Y 386.884,Z 729.378,A -85,B 0,C 180,E1 11827.271,E2 11827.271} C_VEL
LIN {X 0,Y 394.058,Z 695.076,A -85,B 0,C 180,E1 11830.425,E2 11830.425} C_VEL
LIN {X 0,Y 400.339,Z 657.983,A -85,B 0,C 180,E1 11832.809,E2 11832.809} C_VEL
LIN {X 0,Y 403.487,Z 630.827,A -85,B 0,C 180,E1 11834.054,E2 11834.054} C_VEL
LIN {X 0,Y 387.941,Z 596.29,A -85,B 0,C 180,E1 11837.424,E2 11837.424} C_VEL
LIN {X 0,Y 367.259,Z 560.732,A -85,B 0,C 180,E1 11841.529,E2 11841.529} C_VEL
LIN {X 0,Y 361.455,Z 550.745,A -85,B 0,C 180,E1 11842.802,E2 11842.802} C_VEL
LIN {X 0,Y 361.342,Z 549.53,A -85,B 0,C 180,E1 11842.993,E2 11842.993} C_VEL
LIN {X 0,Y 361.334,Z 549.53,A -85,B 0,C 180,E1 11849.909,E2 11849.909} C_VEL
LIN {X 0,Y 361.701,Z 549.53,A -85,B 0,C 180,E1 11857.93,E2 11857.93} C_VEL
LIN {X 0,Y 361.951,Z 549.53,A -85,B 0,C 180,E1 11865.497,E2 11865.497} C_VEL
LIN {X 0,Y 362.468,Z 549.53,A -85,B 0,C 180,E1 11872.807,E2 11872.807} C_VEL
LIN {X 0,Y 362.861,Z 549.53,A -85,B 0,C 180,E1 11879.98,E2 11879.98} C_VEL
LIN {X 0,Y 362.478,Z 549.53,A -85,B 0,C 180,E1 11887.153,E2 11887.153} C_VEL
LIN {X 0,Y 362.131,Z 549.53,A -85,B 0,C 180,E1 11894.455,E2 11894.455} C_VEL
LIN {X 0,Y 361.725,Z 549.53,A -85,B 0,C 180,E1 11902.025,E2 11902.025} C_VEL
LIN {X 0,Y 361.478,Z 549.53,A -85,B 0,C 180,E1 11910.032,E2 11910.032} C_VEL
LIN {X 0,Y 361.325,Z 549.53,A -85,B 0,C 180,E1 11917.483,E2 11917.483} C_VEL
LIN {X 0,Y 361.206,Z 549.53,A -85,B 0,C 180,E1 11924.745,E2 11924.745} C_VEL
LIN {X 0,Y 361.307,Z 549.53,A -85,B 0,C 180,E1 11931.207,E2 11931.207} C_VEL
LIN {X 0,Y 361.39,Z 549.53,A -85,B 0,C 180,E1 11937.122,E2 11937.122} C_VEL
LIN {X 0,Y 361.518,Z 549.53,A -85,B 0,C 180,E1 11942.666,E2 11942.666} C_VEL
LIN {X 0,Y 361.834,Z 550.056,A -85,B 0,C 180,E1 11949.596,E2 11949.596} C_VEL
LIN {X 0,Y 364.668,Z 555.596,A -85,B 0,C 180,E1 11950.23,E2 11950.23} C_VEL
LIN {X 0,Y 382.172,Z 587.12,A -85,B 0,C 180,E1 11954.07,E2 11954.07} C_VEL
LIN {X 0,Y 394.295,Z 617.493,A -85,B 0,C 180,E1 11957.462,E2 11957.462} C_VEL
LIN {X 0,Y 396.118,Z 625.572,A -85,B 0,C 180,E1 11958.277,E2 11958.277} C_VEL
LIN {X 0,Y 390.218,Z 660.867,A -85,B 0,C 180,E1 11960.866,E2 11960.866} C_VEL
LIN {X 0,Y 383.574,Z 692.593,A -85,B 0,C 180,E1 11964.212,E2 11964.212} C_VEL
LIN {X 0,Y 377.035,Z 720.494,A -85,B 0,C 180,E1 11968.309,E2 11968.309} C_VEL
LIN {X 0,Y 371.28,Z 744.389,A -85,B 0,C 180,E1 11973.182,E2 11973.182} C_VEL
LIN {X 0,Y 367.4,Z 761.854,A -85,B 0,C 180,E1 11978.171,E2 11978.171} C_VEL
LIN {X 0,Y 364.758,Z 775.473,A -85,B 0,C 180,E1 11983.861,E2 11983.861} C_VEL
LIN {X 0,Y 363.514,Z 783.442,A -85,B 0,C 180,E1 11989.394,E2 11989.394} C_VEL
LIN {X 0,Y 362.754,Z 786.692,A -85,B 0,C 180,E1 11994.58,E2 11994.58} C_VEL
LIN {X 0,Y 363.099,Z 785.846,A -85,B 0,C 180,E1 11999.913,E2 11999.913} C_VEL
LIN {X 0,Y 364.259,Z 780.448,A -85,B 0,C 180,E1 12005.447,E2 12005.447} C_VEL
LIN {X 0,Y 366.223,Z 769.589,A -85,B 0,C 180,E1 12011.242,E2 12011.242} C_VEL
LIN {X 0,Y 369.878,Z 753.114,A -85,B 0,C 180,E1 12016.877,E2 12016.877} C_VEL
LIN {X 0,Y 375.585,Z 730.724,A -85,B 0,C 180,E1 12022.153,E2 12022.153} C_VEL
LIN {X 0,Y 382.34,Z 704.087,A -85,B 0,C 180,E1 12026.592,E2 12026.592} C_VEL
LIN {X 0,Y 389.242,Z 674.174,A -85,B 0,C 180,E1 12030.192,E2 12030.192} C_VEL
LIN {X 0,Y 396.024,Z 639.119,A -85,B 0,C 180,E1 12033.155,E2 12033.155} C_VEL
LIN {X 0,Y 397.744,Z 625.035,A -85,B 0,C 180,E1 12034.112,E2 12034.112} C_VEL
LIN {X 0,Y 387.04,Z 595.158,A -85,B 0,C 180,E1 12037.683,E2 12037.683} C_VEL
LIN {X 0,Y 372.677,Z 567.746,A -85,B 0,C 180,E1 12041.43,E2 12041.43} C_VEL
LIN {X 0,Y 364.083,Z 554.918,A -85,B 0,C 180,E1 12043.613,E2 12043.613} C_VEL
LIN {X 0,Y 361.929,Z 549.53,A -85,B 0,C 180,E1 12044.3,E2 12044.3} C_VEL
LIN {X 0,Y 362.246,Z 549.53,A -85,B 0,C 180,E1 12050.431,E2 12050.431} C_VEL
LIN {X 0,Y 362.829,Z 549.53,A -85,B 0,C 180,E1 12057.637,E2 12057.637} C_VEL
LIN {X 0,Y 362.626,Z 549.53,A -85,B 0,C 180,E1 12064.793,E2 12064.793} C_VEL
LIN {X 0,Y 362.283,Z 549.53,A -85,B 0,C 180,E1 12072.038,E2 12072.038} C_VEL
LIN {X 0,Y 361.85,Z 549.53,A -85,B 0,C 180,E1 12079.505,E2 12079.505} C_VEL
LIN {X 0,Y 361.646,Z 549.53,A -85,B 0,C 180,E1 12084.678,E2 12084.678} C_VEL
LIN {X 0,Y 361.496,Z 549.53,A -85,B 0,C 180,E1 12090.076,E2 12090.076} C_VEL
LIN {X 0,Y 361.461,Z 550.231,A -85,B 0,C 180,E1 12095.927,E2 12095.927} C_VEL
LIN {X 0,Y 364.182,Z 555.508,A -85,B 0,C 180,E1 12096.7,E2 12096.7} C_VEL
LIN {X 0,Y 377.697,Z 576.544,A -85,B 0,C 180,E1 12099.97,E2 12099.97} C_VEL
LIN {X 0,Y 393.888,Z 606.232,A -85,B 0,C 180,E1 12103.506,E2 12103.506} C_VEL
LIN {X 0,Y 403.845,Z 632.133,A -85,B 0,C 180,E1 12106.033,E2 12106.033} C_VEL
LIN {X 0,Y 398.483,Z 669.403,A -85,B 0,C 180,E1 12107.839,E2 12107.839} C_VEL
LIN {X 0,Y 391.545,Z 706.406,A -85,B 0,C 180,E1 12110.554,E2 12110.554} C_VEL
LIN {X 0,Y 384.105,Z 740.299,A -85,B 0,C 180,E1 12114.069,E2 12114.069} C_VEL
LIN {X 0,Y 376.965,Z 770.593,A -85,B 0,C 180,E1 12118.353,E2 12118.353} C_VEL
LIN {X 0,Y 370.847,Z 797.751,A -85,B 0,C 180,E1 12123.551,E2 12123.551} C_VEL
LIN {X 0,Y 366.485,Z 820.444,A -85,B 0,C 180,E1 12129.515,E2 12129.515} C_VEL
LIN {X 0,Y 364.098,Z 836.618,A -85,B 0,C 180,E1 12135.603,E2 12135.603} C_VEL
LIN {X 0,Y 363.275,Z 846.851,A -85,B 0,C 180,E1 12141.642,E2 12141.642} C_VEL
LIN {X 0,Y 363.153,Z 851.611,A -85,B 0,C 180,E1 12147.62,E2 12147.62} C_VEL
LIN {X 0,Y 363.185,Z 851.664,A -85,B 0,C 180,E1 12152.383,E2 12152.383} C_VEL
LIN {X 0,Y 363.266,Z 847.044,A -85,B 0,C 180,E1 12158.362,E2 12158.362} C_VEL
LIN {X 0,Y 363.46,Z 843.866,A -85,B 0,C 180,E1 12160.624,E2 12160.624} C_VEL
LIN {X 0,Y 361.288,Z 840.532,A -85,B 0,C 180,E1 12162.602,E2 12162.602} C_VEL
LIN {X 0,Y 356.59,Z 834.444,A -85,B 0,C 180,E1 12165.535,E2 12165.535} C_VEL
LIN {X 0,Y 356.59,Z 833.687,A -85,B 0,C 180,E1 12165.869,E2 12165.869} C_VEL
LIN {X 0,Y 359.29,Z 817.135,A -85,B 0,C 180,E1 12171.887,E2 12171.887} C_VEL
LIN {X 0,Y 363.986,Z 795.657,A -85,B 0,C 180,E1 12177.468,E2 12177.468} C_VEL
LIN {X 0,Y 370.421,Z 769.175,A -85,B 0,C 180,E1 12182.531,E2 12182.531} C_VEL
LIN {X 0,Y 378.034,Z 738.141,A -85,B 0,C 180,E1 12186.901,E2 12186.901} C_VEL
LIN {X 0,Y 386.247,Z 701.885,A -85,B 0,C 180,E1 12190.558,E2 12190.558} C_VEL
LIN {X 0,Y 393.177,Z 664.452,A -85,B 0,C 180,E1 12193.167,E2 12193.167} C_VEL
LIN {X 0,Y 396.97,Z 632.899,A -85,B 0,C 180,E1 12194.731,E2 12194.731} C_VEL
LIN {X 0,Y 381.424,Z 598.193,A -85,B 0,C 180,E1 12198.289,E2 12198.289} C_VEL
LIN {X 0,Y 359.737,Z 561.097,A -85,B 0,C 180,E1 12202.8,E2 12202.8} C_VEL
LIN {X 0,Y 353.51,Z 550.934,A -85,B 0,C 180,E1 12204.224,E2 12204.224} C_VEL
LIN {X 0,Y 353.348,Z 549.53,A -85,B 0,C 180,E1 12204.323,E2 12204.323} C_VEL
LIN {X 0,Y 353.448,Z 549.53,A -85,B 0,C 180,E1 12211.974,E2 12211.974} C_VEL
LIN {X 0,Y 353.819,Z 549.53,A -85,B 0,C 180,E1 12219.77,E2 12219.77} C_VEL
LIN {X 0,Y 354.148,Z 549.53,A -85,B 0,C 180,E1 12227.681,E2 12227.681} C_VEL
LIN {X 0,Y 354.697,Z 549.53,A -85,B 0,C 180,E1 12235.1,E2 12235.1} C_VEL
LIN {X 0,Y 354.965,Z 549.53,A -85,B 0,C 180,E1 12239.98,E2 12239.98} C_VEL
LIN {X 0,Y 354.546,Z 549.53,A -85,B 0,C 180,E1 12247.314,E2 12247.314} C_VEL
LIN {X 0,Y 354.196,Z 549.53,A -85,B 0,C 180,E1 12254.786,E2 12254.786} C_VEL
LIN {X 0,Y 353.784,Z 549.53,A -85,B 0,C 180,E1 12262.547,E2 12262.547} C_VEL
LIN {X 0,Y 353.567,Z 549.53,A -85,B 0,C 180,E1 12267.97,E2 12267.97} C_VEL
LIN {X 0,Y 353.47,Z 549.53,A -85,B 0,C 180,E1 12275.79,E2 12275.79} C_VEL
LIN {X 0,Y 353.209,Z 549.53,A -85,B 0,C 180,E1 12283.421,E2 12283.421} C_VEL
LIN {X 0,Y 353.33,Z 549.53,A -85,B 0,C 180,E1 12290.194,E2 12290.194} C_VEL
LIN {X 0,Y 353.445,Z 549.53,A -85,B 0,C 180,E1 12296.285,E2 12296.285} C_VEL
LIN {X 0,Y 353.58,Z 549.53,A -85,B 0,C 180,E1 12303.595,E2 12303.595} C_VEL
LIN {X 0,Y 353.854,Z 549.53,A -85,B 0,C 180,E1 12308.167,E2 12308.167} C_VEL
LIN {X 0,Y 356.226,Z 555.184,A -85,B 0,C 180,E1 12308.79,E2 12308.79} C_VEL
LIN {X 0,Y 373.605,Z 585.165,A -85,B 0,C 180,E1 12312.736,E2 12312.736} C_VEL
LIN {X 0,Y 386.803,Z 616.759,A -85,B 0,C 180,E1 12316.461,E2 12316.461} C_VEL
LIN {X 0,Y 389.691,Z 627.788,A -85,B 0,C 180,E1 12317.663,E2 12317.663} C_VEL
LIN {X 0,Y 383.345,Z 663.445,A -85,B 0,C 180,E1 12320.368,E2 12320.368} C_VEL
LIN {X 0,Y 376.668,Z 693.943,A -85,B 0,C 180,E1 12323.673,E2 12323.673} C_VEL
LIN {X 0,Y 369.773,Z 722.077,A -85,B 0,C 180,E1 12327.903,E2 12327.903} C_VEL
LIN {X 0,Y 363.863,Z 745.27,A -85,B 0,C 180,E1 12332.757,E2 12332.757} C_VEL
LIN {X 0,Y 359.549,Z 763.751,A -85,B 0,C 180,E1 12338.232,E2 12338.232} C_VEL
LIN {X 0,Y 356.992,Z 776.3,A -85,B 0,C 180,E1 12343.68,E2 12343.68} C_VEL
LIN {X 0,Y 355.966,Z 782.826,A -85,B 0,C 180,E1 12348.024,E2 12348.024} C_VEL
LIN {X 0,Y 355.088,Z 786.623,A -85,B 0,C 180,E1 12352.485,E2 12352.485} C_VEL
LIN {X 0,Y 354.948,Z 787.427,A -85,B 0,C 180,E1 12357.88,E2 12357.88} C_VEL
LIN {X 0,Y 355.995,Z 783.859,A -85,B 0,C 180,E1 12363.437,E2 12363.437} C_VEL
LIN {X 0,Y 357.524,Z 775.293,A -85,B 0,C 180,E1 12369.278,E2 12369.278} C_VEL
LIN {X 0,Y 360.855,Z 760.465,A -85,B 0,C 180,E1 12375.306,E2 12375.306} C_VEL
LIN {X 0,Y 365.783,Z 741.552,A -85,B 0,C 180,E1 12380.535,E2 12380.535} C_VEL
LIN {X 0,Y 372.702,Z 716.19,A -85,B 0,C 180,E1 12385.503,E2 12385.503} C_VEL
LIN {X 0,Y 379.978,Z 687.335,A -85,B 0,C 180,E1 12389.524,E2 12389.524} C_VEL
LIN {X 0,Y 387.153,Z 654.882,A -85,B 0,C 180,E1 12392.745,E2 12392.745} C_VEL
LIN {X 0,Y 391.461,Z 627.665,A -85,B 0,C 180,E1 12394.761,E2 12394.761} C_VEL
LIN {X 0,Y 380.704,Z 597.143,A -85,B 0,C 180,E1 12398.593,E2 12398.593} C_VEL
LIN {X 0,Y 367.465,Z 571.901,A -85,B 0,C 180,E1 12402.28,E2 12402.28} C_VEL
LIN {X 0,Y 356.901,Z 555.6,A -85,B 0,C 180,E1 12405.188,E2 12405.188} C_VEL
LIN {X 0,Y 354.099,Z 550.197,A -85,B 0,C 180,E1 12406.076,E2 12406.076} C_VEL
LIN {X 0,Y 354.539,Z 549.53,A -85,B 0,C 180,E1 12413.116,E2 12413.116} C_VEL
LIN {X 0,Y 354.967,Z 549.53,A -85,B 0,C 180,E1 12420.02,E2 12420.02} C_VEL
LIN {X 0,Y 354.544,Z 549.53,A -85,B 0,C 180,E1 12427.355,E2 12427.355} C_VEL
LIN {X 0,Y 354.218,Z 549.53,A -85,B 0,C 180,E1 12434.827,E2 12434.827} C_VEL
LIN {X 0,Y 353.776,Z 549.53,A -85,B 0,C 180,E1 12442.591,E2 12442.591} C_VEL
LIN {X 0,Y 353.568,Z 549.53,A -85,B 0,C 180,E1 12448.016,E2 12448.016} C_VEL
LIN {X 0,Y 353.461,Z 550.175,A -85,B 0,C 180,E1 12454.036,E2 12454.036} C_VEL
LIN {X 0,Y 356.041,Z 555.414,A -85,B 0,C 180,E1 12454.861,E2 12454.861} C_VEL
LIN {X 0,Y 358.848,Z 559.31,A -85,B 0,C 180,E1 12455.651,E2 12455.651} C_VEL
LIN {X 0,Y 372.362,Z 579.732,A -85,B 0,C 180,E1 12459.091,E2 12459.091} C_VEL
LIN {X 0,Y 388.91,Z 611.184,A -85,B 0,C 180,E1 12462.969,E2 12462.969} C_VEL
LIN {X 0,Y 397.662,Z 634.451,A -85,B 0,C 180,E1 12465.364,E2 12465.364} C_VEL
LIN {X 0,Y 391.737,Z 672.93,A -85,B 0,C 180,E1 12467.329,E2 12467.329} C_VEL
LIN {X 0,Y 384.303,Z 710.102,A -85,B 0,C 180,E1 12470.196,E2 12470.196} C_VEL
LIN {X 0,Y 376.049,Z 745.305,A -85,B 0,C 180,E1 12474.067,E2 12474.067} C_VEL
LIN {X 0,Y 368.677,Z 775.344,A -85,B 0,C 180,E1 12478.64,E2 12478.64} C_VEL
LIN {X 0,Y 362.604,Z 800.83,A -85,B 0,C 180,E1 12483.879,E2 12483.879} C_VEL
LIN {X 0,Y 358.46,Z 821.51,A -85,B 0,C 180,E1 12489.68,E2 12489.68} C_VEL
LIN {X 0,Y 356.136,Z 836.947,A -85,B 0,C 180,E1 12495.824,E2 12495.824} C_VEL
LIN {X 0,Y 355.401,Z 846.123,A -85,B 0,C 180,E1 12501.456,E2 12501.456} C_VEL
LIN {X 0,Y 355.299,Z 850.903,A -85,B 0,C 180,E1 12507.568,E2 12507.568} C_VEL
LIN {X 0,Y 355.331,Z 850.961,A -85,B 0,C 180,E1 12512.436,E2 12512.436} C_VEL
LIN {X 0,Y 355.387,Z 846.334,A -85,B 0,C 180,E1 12518.548,E2 12518.548} C_VEL
LIN {X 0,Y 356.287,Z 836.239,A -85,B 0,C 180,E1 12524.724,E2 12524.724} C_VEL
LIN {X 0,Y 356.59,Z 833.687,A -85,B 0,C 180,E1 12525.869,E2 12525.869} C_VEL
LIN {X 0,Y 353.593,Z 827.468,A -85,B 0,C 180,E1 12528.467,E2 12528.467} C_VEL
LIN {X 0,Y 350.901,Z 820.48,A -85,B 0,C 180,E1 12531.06,E2 12531.06} C_VEL
LIN {X 0,Y 355.821,Z 798.418,A -85,B 0,C 180,E1 12537.253,E2 12537.253} C_VEL
LIN {X 0,Y 362.747,Z 771.152,A -85,B 0,C 180,E1 12542.74,E2 12542.74} C_VEL
LIN {X 0,Y 370.369,Z 741.409,A -85,B 0,C 180,E1 12547.124,E2 12547.124} C_VEL
LIN {X 0,Y 378.396,Z 707.849,A -85,B 0,C 180,E1 12550.724,E2 12550.724} C_VEL
LIN {X 0,Y 385.446,Z 673.105,A -85,B 0,C 180,E1 12553.377,E2 12553.377} C_VEL
LIN {X 0,Y 390.632,Z 635.658,A -85,B 0,C 180,E1 12555.369,E2 12555.369} C_VEL
LIN {X 0,Y 375.622,Z 601.387,A -85,B 0,C 180,E1 12559.041,E2 12559.041} C_VEL
LIN {X 0,Y 355.07,Z 566.285,A -85,B 0,C 180,E1 12563.473,E2 12563.473} C_VEL
LIN {X 0,Y 345.653,Z 551.48,A -85,B 0,C 180,E1 12565.714,E2 12565.714} C_VEL
LIN {X 0,Y 345.402,Z 549.53,A -85,B 0,C 180,E1 12565.993,E2 12565.993} C_VEL
LIN {X 0,Y 345.638,Z 549.53,A -85,B 0,C 180,E1 12574.097,E2 12574.097} C_VEL
LIN {X 0,Y 345.986,Z 549.53,A -85,B 0,C 180,E1 12582.206,E2 12582.206} C_VEL
LIN {X 0,Y 346.359,Z 549.53,A -85,B 0,C 180,E1 12589.945,E2 12589.945} C_VEL
LIN {X 0,Y 347.055,Z 549.53,A -85,B 0,C 180,E1 12597.488,E2 12597.488} C_VEL
LIN {X 0,Y 346.814,Z 549.53,A -85,B 0,C 180,E1 12604.97,E2 12604.97} C_VEL
LIN {X 0,Y 346.388,Z 549.53,A -85,B 0,C 180,E1 12612.557,E2 12612.557} C_VEL
LIN {X 0,Y 345.924,Z 549.53,A -85,B 0,C 180,E1 12620.398,E2 12620.398} C_VEL
LIN {X 0,Y 345.709,Z 549.53,A -85,B 0,C 180,E1 12625.851,E2 12625.851} C_VEL
LIN {X 0,Y 345.53,Z 549.53,A -85,B 0,C 180,E1 12633.921,E2 12633.921} C_VEL
LIN {X 0,Y 345.251,Z 549.53,A -85,B 0,C 180,E1 12640.927,E2 12640.927} C_VEL
LIN {X 0,Y 345.226,Z 549.53,A -85,B 0,C 180,E1 12647.949,E2 12647.949} C_VEL
LIN {X 0,Y 345.521,Z 549.53,A -85,B 0,C 180,E1 12655.404,E2 12655.404} C_VEL
LIN {X 0,Y 345.562,Z 549.53,A -85,B 0,C 180,E1 12661.29,E2 12661.29} C_VEL
LIN {X 0,Y 345.801,Z 549.53,A -85,B 0,C 180,E1 12666.672,E2 12666.672} C_VEL
LIN {X 0,Y 348.261,Z 555.169,A -85,B 0,C 180,E1 12667.353,E2 12667.353} C_VEL
LIN {X 0,Y 365.765,Z 584.59,A -85,B 0,C 180,E1 12671.501,E2 12671.501} C_VEL
LIN {X 0,Y 379.168,Z 615.819,A -85,B 0,C 180,E1 12675.386,E2 12675.386} C_VEL
LIN {X 0,Y 383.064,Z 630.819,A -85,B 0,C 180,E1 12677.085,E2 12677.085} C_VEL
LIN {X 0,Y 376.804,Z 664.717,A -85,B 0,C 180,E1 12679.733,E2 12679.733} C_VEL
LIN {X 0,Y 369.81,Z 695.283,A -85,B 0,C 180,E1 12683.114,E2 12683.114} C_VEL
LIN {X 0,Y 362.338,Z 724.311,A -85,B 0,C 180,E1 12687.611,E2 12687.611} C_VEL
LIN {X 0,Y 356.053,Z 747.748,A -85,B 0,C 180,E1 12692.736,E2 12692.736} C_VEL
LIN {X 0,Y 351.731,Z 765.439,A -85,B 0,C 180,E1 12698.217,E2 12698.217} C_VEL
LIN {X 0,Y 349.07,Z 778.03,A -85,B 0,C 180,E1 12703.996,E2 12703.996} C_VEL
LIN {X 0,Y 347.896,Z 784.703,A -85,B 0,C 180,E1 12708.981,E2 12708.981} C_VEL
LIN {X 0,Y 346.999,Z 788.041,A -85,B 0,C 180,E1 12714.124,E2 12714.124} C_VEL
LIN {X 0,Y 347.3,Z 787.492,A -85,B 0,C 180,E1 12719.723,E2 12719.723} C_VEL
LIN {X 0,Y 348.685,Z 781.926,A -85,B 0,C 180,E1 12725.894,E2 12725.894} C_VEL
LIN {X 0,Y 350.866,Z 771.514,A -85,B 0,C 180,E1 12731.775,E2 12731.775} C_VEL
LIN {X 0,Y 354.946,Z 755.343,A -85,B 0,C 180,E1 12737.623,E2 12737.623} C_VEL
LIN {X 0,Y 361.073,Z 733.924,A -85,B 0,C 180,E1 12742.967,E2 12742.967} C_VEL
LIN {X 0,Y 368.703,Z 706.821,A -85,B 0,C 180,E1 12747.733,E2 12747.733} C_VEL
LIN {X 0,Y 376.092,Z 677.919,A -85,B 0,C 180,E1 12751.379,E2 12751.379} C_VEL
LIN {X 0,Y 383.263,Z 644.612,A -85,B 0,C 180,E1 12754.363,E2 12754.363} C_VEL
LIN {X 0,Y 385.282,Z 630.618,A -85,B 0,C 180,E1 12755.404,E2 12755.404} C_VEL
LIN {X 0,Y 375.214,Z 601.07,A -85,B 0,C 180,E1 12759.265,E2 12759.265} C_VEL
LIN {X 0,Y 361.965,Z 574.825,A -85,B 0,C 180,E1 12763.286,E2 12763.286} C_VEL
LIN {X 0,Y 349.273,Z 555.778,A -85,B 0,C 180,E1 12767.073,E2 12767.073} C_VEL
LIN {X 0,Y 346.377,Z 550.733,A -85,B 0,C 180,E1 12768.078,E2 12768.078} C_VEL
LIN {X 0,Y 346.297,Z 549.53,A -85,B 0,C 180,E1 12768.436,E2 12768.436} C_VEL
LIN {X 0,Y 346.8,Z 549.53,A -85,B 0,C 180,E1 12775.03,E2 12775.03} C_VEL
LIN {X 0,Y 347.063,Z 549.53,A -85,B 0,C 180,E1 12780.147,E2 12780.147} C_VEL
LIN {X 0,Y 346.632,Z 549.53,A -85,B 0,C 180,E1 12787.523,E2 12787.523} C_VEL
LIN {X 0,Y 346.248,Z 549.53,A -85,B 0,C 180,E1 12795.176,E2 12795.176} C_VEL
LIN {X 0,Y 345.785,Z 549.53,A -85,B 0,C 180,E1 12803.143,E2 12803.143} C_VEL
LIN {X 0,Y 345.551,Z 549.53,A -85,B 0,C 180,E1 12809.148,E2 12809.148} C_VEL
LIN {X 0,Y 345.539,Z 549.658,A -85,B 0,C 180,E1 12811.898,E2 12811.898} C_VEL
LIN {X 0,Y 347.585,Z 554.851,A -85,B 0,C 180,E1 12812.683,E2 12812.683} C_VEL
LIN {X 0,Y 350.476,Z 558.2,A -85,B 0,C 180,E1 12813.582,E2 12813.582} C_VEL
LIN {X 0,Y 365.276,Z 580.229,A -85,B 0,C 180,E1 12817.725,E2 12817.725} C_VEL
LIN {X 0,Y 381.668,Z 611.045,A -85,B 0,C 180,E1 12821.839,E2 12821.839} C_VEL
LIN {X 0,Y 391.557,Z 636.788,A -85,B 0,C 180,E1 12824.678,E2 12824.678} C_VEL
LIN {X 0,Y 385.153,Z 675.843,A -85,B 0,C 180,E1 12826.758,E2 12826.758} C_VEL
LIN {X 0,Y 377.12,Z 713.379,A -85,B 0,C 180,E1 12829.8,E2 12829.8} C_VEL
LIN {X 0,Y 368.572,Z 747.74,A -85,B 0,C 180,E1 12833.767,E2 12833.767} C_VEL
LIN {X 0,Y 360.858,Z 777.638,A -85,B 0,C 180,E1 12838.537,E2 12838.537} C_VEL
LIN {X 0,Y 354.55,Z 802.571,A -85,B 0,C 180,E1 12843.926,E2 12843.926} C_VEL
LIN {X 0,Y 350.417,Z 822.579,A -85,B 0,C 180,E1 12849.85,E2 12849.85} C_VEL
LIN {X 0,Y 348.147,Z 837.576,A -85,B 0,C 180,E1 12856.21,E2 12856.21} C_VEL
LIN {X 0,Y 347.552,Z 845.4,A -85,B 0,C 180,E1 12861.261,E2 12861.261} C_VEL
LIN {X 0,Y 347.444,Z 850.196,A -85,B 0,C 180,E1 12867.513,E2 12867.513} C_VEL
LIN {X 0,Y 347.46,Z 850.232,A -85,B 0,C 180,E1 12872.548,E2 12872.548} C_VEL
LIN {X 0,Y 347.504,Z 845.615,A -85,B 0,C 180,E1 12878.744,E2 12878.744} C_VEL
LIN {X 0,Y 348.468,Z 835.501,A -85,B 0,C 180,E1 12885.062,E2 12885.062} C_VEL
LIN {X 0,Y 350.901,Z 820.48,A -85,B 0,C 180,E1 12891.06,E2 12891.06} C_VEL
LIN {X 0,Y 348.671,Z 812.902,A -85,B 0,C 180,E1 12893.624,E2 12893.624} C_VEL
LIN {X 0,Y 346.737,Z 804.405,A -85,B 0,C 180,E1 12896.141,E2 12896.141} C_VEL
LIN {X 0,Y 353.27,Z 779.433,A -85,B 0,C 180,E1 12901.773,E2 12901.773} C_VEL
LIN {X 0,Y 361.015,Z 751.091,A -85,B 0,C 180,E1 12906.458,E2 12906.458} C_VEL
LIN {X 0,Y 369.174,Z 719.705,A -85,B 0,C 180,E1 12910.269,E2 12910.269} C_VEL
LIN {X 0,Y 377.035,Z 684.341,A -85,B 0,C 180,E1 12913.356,E2 12913.356} C_VEL
LIN {X 0,Y 383.503,Z 647.72,A -85,B 0,C 180,E1 12915.537,E2 12915.537} C_VEL
LIN {X 0,Y 384.292,Z 638.246,A -85,B 0,C 180,E1 12916.041,E2 12916.041} C_VEL
LIN {X 0,Y 369.526,Z 604.095,A -85,B 0,C 180,E1 12919.862,E2 12919.862} C_VEL
LIN {X 0,Y 348.629,Z 568.077,A -85,B 0,C 180,E1 12924.609,E2 12924.609} C_VEL
LIN {X 0,Y 337.68,Z 551.446,A -85,B 0,C 180,E1 12927.347,E2 12927.347} C_VEL
LIN {X 0,Y 337.466,Z 549.53,A -85,B 0,C 180,E1 12927.531,E2 12927.531} C_VEL
LIN {X 0,Y 337.819,Z 549.53,A -85,B 0,C 180,E1 12936.278,E2 12936.278} C_VEL
LIN {X 0,Y 338.02,Z 549.53,A -85,B 0,C 180,E1 12941.772,E2 12941.772} C_VEL
LIN {X 0,Y 338.413,Z 549.53,A -85,B 0,C 180,E1 12949.706,E2 12949.706} C_VEL
LIN {X 0,Y 339.136,Z 549.53,A -85,B 0,C 180,E1 12957.429,E2 12957.429} C_VEL
LIN {X 0,Y 339.044,Z 549.53,A -85,B 0,C 180,E1 12962.529,E2 12962.529} C_VEL
LIN {X 0,Y 338.526,Z 549.53,A -85,B 0,C 180,E1 12970.247,E2 12970.247} C_VEL
LIN {X 0,Y 338.091,Z 549.53,A -85,B 0,C 180,E1 12978.179,E2 12978.179} C_VEL
LIN {X 0,Y 337.856,Z 549.53,A -85,B 0,C 180,E1 12983.673,E2 12983.673} C_VEL
LIN {X 0,Y 337.634,Z 549.53,A -85,B 0,C 180,E1 12991.874,E2 12991.874} C_VEL
LIN {X 0,Y 337.387,Z 549.53,A -85,B 0,C 180,E1 12998.73,E2 12998.73} C_VEL
LIN {X 0,Y 337.303,Z 549.53,A -85,B 0,C 180,E1 13005.665,E2 13005.665} C_VEL
LIN {X 0,Y 337.436,Z 549.53,A -85,B 0,C 180,E1 13013.552,E2 13013.552} C_VEL
LIN {X 0,Y 337.633,Z 549.53,A -85,B 0,C 180,E1 13020.55,E2 13020.55} C_VEL
LIN {X 0,Y 337.779,Z 549.53,A -85,B 0,C 180,E1 13025.094,E2 13025.094} C_VEL
LIN {X 0,Y 340.031,Z 554.994,A -85,B 0,C 180,E1 13025.752,E2 13025.752} C_VEL
LIN {X 0,Y 355.647,Z 580.106,A -85,B 0,C 180,E1 13029.635,E2 13029.635} C_VEL
LIN {X 0,Y 369.407,Z 609.394,A -85,B 0,C 180,E1 13033.549,E2 13033.549} C_VEL
LIN {X 0,Y 376.811,Z 632.16,A -85,B 0,C 180,E1 13036.384,E2 13036.384} C_VEL
LIN {X 0,Y 370.172,Z 666.543,A -85,B 0,C 180,E1 13039.131,E2 13039.131} C_VEL
LIN {X 0,Y 362.698,Z 697.63,A -85,B 0,C 180,E1 13042.663,E2 13042.663} C_VEL
LIN {X 0,Y 355.116,Z 725.741,A -85,B 0,C 180,E1 13047.163,E2 13047.163} C_VEL
LIN {X 0,Y 348.77,Z 748.185,A -85,B 0,C 180,E1 13052.168,E2 13052.168} C_VEL
LIN {X 0,Y 344.039,Z 766.533,A -85,B 0,C 180,E1 13057.981,E2 13057.981} C_VEL
LIN {X 0,Y 341.127,Z 779.81,A -85,B 0,C 180,E1 13064.398,E2 13064.398} C_VEL
LIN {X 0,Y 339.93,Z 785.979,A -85,B 0,C 180,E1 13069.445,E2 13069.445} C_VEL
LIN {X 0,Y 339.189,Z 788.562,A -85,B 0,C 180,E1 13073.601,E2 13073.601} C_VEL
LIN {X 0,Y 339.362,Z 788.402,A -85,B 0,C 180,E1 13079.281,E2 13079.281} C_VEL
LIN {X 0,Y 340.638,Z 783.828,A -85,B 0,C 180,E1 13085.16,E2 13085.16} C_VEL
LIN {X 0,Y 342.994,Z 773.411,A -85,B 0,C 180,E1 13091.636,E2 13091.636} C_VEL
LIN {X 0,Y 347.187,Z 757.724,A -85,B 0,C 180,E1 13097.634,E2 13097.634} C_VEL
LIN {X 0,Y 353.562,Z 736.367,A -85,B 0,C 180,E1 13103.21,E2 13103.21} C_VEL
LIN {X 0,Y 361.487,Z 710.01,A -85,B 0,C 180,E1 13108.066,E2 13108.066} C_VEL
LIN {X 0,Y 369.62,Z 679.716,A -85,B 0,C 180,E1 13112.014,E2 13112.014} C_VEL
LIN {X 0,Y 377.228,Z 646.002,A -85,B 0,C 180,E1 13115.103,E2 13115.103} C_VEL
LIN {X 0,Y 379.012,Z 633.261,A -85,B 0,C 180,E1 13116.097,E2 13116.097} C_VEL
LIN {X 0,Y 369.757,Z 604.951,A -85,B 0,C 180,E1 13119.966,E2 13119.966} C_VEL
LIN {X 0,Y 357.636,Z 580.272,A -85,B 0,C 180,E1 13123.95,E2 13123.95} C_VEL
LIN {X 0,Y 345.557,Z 561.71,A -85,B 0,C 180,E1 13127.82,E2 13127.82} C_VEL
LIN {X 0,Y 341.828,Z 556.041,A -85,B 0,C 180,E1 13129.153,E2 13129.153} C_VEL
LIN {X 0,Y 338.602,Z 550.963,A -85,B 0,C 180,E1 13130.403,E2 13130.403} C_VEL
LIN {X 0,Y 338.496,Z 549.53,A -85,B 0,C 180,E1 13130.724,E2 13130.724} C_VEL
LIN {X 0,Y 339.115,Z 549.53,A -85,B 0,C 180,E1 13137.471,E2 13137.471} C_VEL
LIN {X 0,Y 339.027,Z 549.53,A -85,B 0,C 180,E1 13142.572,E2 13142.572} C_VEL
LIN {X 0,Y 338.524,Z 549.53,A -85,B 0,C 180,E1 13150.29,E2 13150.29} C_VEL
LIN {X 0,Y 338.3,Z 549.53,A -85,B 0,C 180,E1 13155.542,E2 13155.542} C_VEL
LIN {X 0,Y 337.945,Z 549.53,A -85,B 0,C 180,E1 13160.947,E2 13160.947} C_VEL
LIN {X 0,Y 337.653,Z 549.53,A -85,B 0,C 180,E1 13169.096,E2 13169.096} C_VEL
LIN {X 0,Y 337.687,Z 550.511,A -85,B 0,C 180,E1 13169.514,E2 13169.514} C_VEL
LIN {X 0,Y 340.5,Z 555.663,A -85,B 0,C 180,E1 13170.657,E2 13170.657} C_VEL
LIN {X 0,Y 342.847,Z 558.404,A -85,B 0,C 180,E1 13171.488,E2 13171.488} C_VEL
LIN {X 0,Y 356.399,Z 578.185,A -85,B 0,C 180,E1 13175.748,E2 13175.748} C_VEL
LIN {X 0,Y 371.593,Z 604.829,A -85,B 0,C 180,E1 13179.855,E2 13179.855} C_VEL
LIN {X 0,Y 384.064,Z 635.094,A -85,B 0,C 180,E1 13183.511,E2 13183.511} C_VEL
LIN {X 0,Y 385.217,Z 640.965,A -85,B 0,C 180,E1 13184.049,E2 13184.049} C_VEL
LIN {X 0,Y 378.512,Z 678.878,A -85,B 0,C 180,E1 13186.196,E2 13186.196} C_VEL
LIN {X 0,Y 370.544,Z 714.067,A -85,B 0,C 180,E1 13189.138,E2 13189.138} C_VEL
LIN {X 0,Y 361.912,Z 746.959,A -85,B 0,C 180,E1 13192.997,E2 13192.997} C_VEL
LIN {X 0,Y 353.861,Z 776.601,A -85,B 0,C 180,E1 13197.792,E2 13197.792} C_VEL
LIN {X 0,Y 347.109,Z 802.134,A -85,B 0,C 180,E1 13203.417,E2 13203.417} C_VEL
LIN {X 0,Y 342.755,Z 821.814,A -85,B 0,C 180,E1 13209.38,E2 13209.38} C_VEL
LIN {X 0,Y 340.344,Z 836.836,A -85,B 0,C 180,E1 13215.888,E2 13215.888} C_VEL
LIN {X 0,Y 339.698,Z 844.677,A -85,B 0,C 180,E1 13221.057,E2 13221.057} C_VEL
LIN {X 0,Y 339.56,Z 849.488,A -85,B 0,C 180,E1 13227.455,E2 13227.455} C_VEL
LIN {X 0,Y 339.586,Z 849.548,A -85,B 0,C 180,E1 13232.549,E2 13232.549} C_VEL
LIN {X 0,Y 339.652,Z 844.897,A -85,B 0,C 180,E1 13238.948,E2 13238.948} C_VEL
LIN {X 0,Y 340.656,Z 834.76,A -85,B 0,C 180,E1 13245.415,E2 13245.415} C_VEL
LIN {X 0,Y 343.387,Z 819.022,A -85,B 0,C 180,E1 13251.793,E2 13251.793} C_VEL
LIN {X 0,Y 346.737,Z 804.405,A -85,B 0,C 180,E1 13256.141,E2 13256.141} C_VEL
LIN {X 0,Y 345.202,Z 795.357,A -85,B 0,C 180,E1 13258.619,E2 13258.619} C_VEL
LIN {X 0,Y 344.265,Z 785.616,A -85,B 0,C 180,E1 13261.041,E2 13261.041} C_VEL
LIN {X 0,Y 352.061,Z 758.224,A -85,B 0,C 180,E1 13266.034,E2 13266.034} C_VEL
LIN {X 0,Y 360.741,Z 726.696,A -85,B 0,C 180,E1 13270.225,E2 13270.225} C_VEL
LIN {X 0,Y 369.38,Z 691.145,A -85,B 0,C 180,E1 13273.599,E2 13273.599} C_VEL
LIN {X 0,Y 376.904,Z 652.035,A -85,B 0,C 180,E1 13276.112,E2 13276.112} C_VEL
LIN {X 0,Y 377.975,Z 640.71,A -85,B 0,C 180,E1 13276.745,E2 13276.745} C_VEL
LIN {X 0,Y 363.454,Z 606.779,A -85,B 0,C 180,E1 13280.702,E2 13280.702} C_VEL
LIN {X 0,Y 344.361,Z 573.664,A -85,B 0,C 180,E1 13285.257,E2 13285.257} C_VEL
LIN {X 0,Y 331.541,Z 554.757,A -85,B 0,C 180,E1 13288.569,E2 13288.569} C_VEL
LIN {X 0,Y 329.541,Z 549.53,A -85,B 0,C 180,E1 13289.303,E2 13289.303} C_VEL
LIN {X 0,Y 329.92,Z 549.53,A -85,B 0,C 180,E1 13296.179,E2 13296.179} C_VEL
LIN {X 0,Y 330.187,Z 549.53,A -85,B 0,C 180,E1 13304.066,E2 13304.066} C_VEL
LIN {X 0,Y 330.709,Z 549.53,A -85,B 0,C 180,E1 13312.112,E2 13312.112} C_VEL
LIN {X 0,Y 331.216,Z 549.53,A -85,B 0,C 180,E1 13317.368,E2 13317.368} C_VEL
LIN {X 0,Y 331.141,Z 549.53,A -85,B 0,C 180,E1 13322.59,E2 13322.59} C_VEL
LIN {X 0,Y 330.611,Z 549.53,A -85,B 0,C 180,E1 13330.495,E2 13330.495} C_VEL
LIN {X 0,Y 330.142,Z 549.53,A -85,B 0,C 180,E1 13338.633,E2 13338.633} C_VEL
LIN {X 0,Y 329.865,Z 549.53,A -85,B 0,C 180,E1 13344.283,E2 13344.283} C_VEL
LIN {X 0,Y 329.694,Z 549.53,A -85,B 0,C 180,E1 13350.197,E2 13350.197} C_VEL
LIN {X 0,Y 329.547,Z 549.53,A -85,B 0,C 180,E1 13356.495,E2 13356.495} C_VEL
LIN {X 0,Y 329.375,Z 549.53,A -85,B 0,C 180,E1 13363.367,E2 13363.367} C_VEL
LIN {X 0,Y 329.465,Z 549.53,A -85,B 0,C 180,E1 13371.084,E2 13371.084} C_VEL
LIN {X 0,Y 329.553,Z 549.53,A -85,B 0,C 180,E1 13376.667,E2 13376.667} C_VEL
LIN {X 0,Y 329.832,Z 549.582,A -85,B 0,C 180,E1 13383.403,E2 13383.403} C_VEL
LIN {X 0,Y 332.003,Z 554.992,A -85,B 0,C 180,E1 13384.08,E2 13384.08} C_VEL
LIN {X 0,Y 347.536,Z 579.12,A -85,B 0,C 180,E1 13388.153,E2 13388.153} C_VEL
LIN {X 0,Y 361.828,Z 608.622,A -85,B 0,C 180,E1 13392.337,E2 13392.337} C_VEL
LIN {X 0,Y 370.321,Z 634.238,A -85,B 0,C 180,E1 13395.686,E2 13395.686} C_VEL
LIN {X 0,Y 363.324,Z 669.454,A -85,B 0,C 180,E1 13398.609,E2 13398.609} C_VEL
LIN {X 0,Y 355.284,Z 701.115,A -85,B 0,C 180,E1 13402.371,E2 13402.371} C_VEL
LIN {X 0,Y 347.614,Z 728.09,A -85,B 0,C 180,E1 13406.878,E2 13406.878} C_VEL
LIN {X 0,Y 340.904,Z 750.965,A -85,B 0,C 180,E1 13412.218,E2 13412.218} C_VEL
LIN {X 0,Y 336.061,Z 768.922,A -85,B 0,C 180,E1 13418.258,E2 13418.258} C_VEL
LIN {X 0,Y 333.421,Z 780.195,A -85,B 0,C 180,E1 13423.93,E2 13423.93} C_VEL
LIN {X 0,Y 331.959,Z 787.242,A -85,B 0,C 180,E1 13429.932,E2 13429.932} C_VEL
LIN {X 0,Y 331.238,Z 789.51,A -85,B 0,C 180,E1 13434.42,E2 13434.42} C_VEL
LIN {X 0,Y 331.613,Z 788.799,A -85,B 0,C 180,E1 13440.229,E2 13440.229} C_VEL
LIN {X 0,Y 333.053,Z 783.801,A -85,B 0,C 180,E1 13446.084,E2 13446.084} C_VEL
LIN {X 0,Y 335.762,Z 772.609,A -85,B 0,C 180,E1 13452.743,E2 13452.743} C_VEL
LIN {X 0,Y 340.544,Z 756.194,A -85,B 0,C 180,E1 13458.874,E2 13458.874} C_VEL
LIN {X 0,Y 347.349,Z 734.745,A -85,B 0,C 180,E1 13464.389,E2 13464.389} C_VEL
LIN {X 0,Y 355.874,Z 707.444,A -85,B 0,C 180,E1 13469.291,E2 13469.291} C_VEL
LIN {X 0,Y 363.99,Z 678.492,A -85,B 0,C 180,E1 13473.006,E2 13473.006} C_VEL
LIN {X 0,Y 371.921,Z 644.462,A -85,B 0,C 180,E1 13476.09,E2 13476.09} C_VEL
LIN {X 0,Y 373.057,Z 636.821,A -85,B 0,C 180,E1 13476.688,E2 13476.688} C_VEL
LIN {X 0,Y 364.39,Z 608.922,A -85,B 0,C 180,E1 13480.678,E2 13480.678} C_VEL
LIN {X 0,Y 353.104,Z 585.325,A -85,B 0,C 180,E1 13484.692,E2 13484.692} C_VEL
LIN {X 0,Y 339.5,Z 563.262,A -85,B 0,C 180,E1 13489.519,E2 13489.519} C_VEL
LIN {X 0,Y 334.122,Z 556.055,A -85,B 0,C 180,E1 13491.666,E2 13491.666} C_VEL
LIN {X 0,Y 330.919,Z 551.012,A -85,B 0,C 180,E1 13493.149,E2 13493.149} C_VEL
LIN {X 0,Y 330.811,Z 549.53,A -85,B 0,C 180,E1 13493.475,E2 13493.475} C_VEL
LIN {X 0,Y 331.336,Z 549.53,A -85,B 0,C 180,E1 13500.022,E2 13500.022} C_VEL
LIN {X 0,Y 330.76,Z 549.53,A -85,B 0,C 180,E1 13507.887,E2 13507.887} C_VEL
LIN {X 0,Y 330.324,Z 549.53,A -85,B 0,C 180,E1 13515.927,E2 13515.927} C_VEL
LIN {X 0,Y 329.853,Z 549.53,A -85,B 0,C 180,E1 13524.331,E2 13524.331} C_VEL
LIN {X 0,Y 329.845,Z 550.093,A -85,B 0,C 180,E1 13526.599,E2 13526.599} C_VEL
LIN {X 0,Y 332.117,Z 555.177,A -85,B 0,C 180,E1 13527.774,E2 13527.774} C_VEL
LIN {X 0,Y 335.05,Z 558.118,A -85,B 0,C 180,E1 13528.987,E2 13528.987} C_VEL
LIN {X 0,Y 345.235,Z 572.833,A -85,B 0,C 180,E1 13532.765,E2 13532.765} C_VEL
LIN {X 0,Y 357.871,Z 592.347,A -85,B 0,C 180,E1 13536.608,E2 13536.608} C_VEL
LIN {X 0,Y 372.213,Z 621.853,A -85,B 0,C 180,E1 13540.838,E2 13540.838} C_VEL
LIN {X 0,Y 379.259,Z 642.651,A -85,B 0,C 180,E1 13543.298,E2 13543.298} C_VEL
LIN {X 0,Y 372.423,Z 679.416,A -85,B 0,C 180,E1 13545.43,E2 13545.43} C_VEL
LIN {X 0,Y 364.017,Z 714.76,A -85,B 0,C 180,E1 13548.453,E2 13548.453} C_VEL
LIN {X 0,Y 355.181,Z 746.875,A -85,B 0,C 180,E1 13552.299,E2 13552.299} C_VEL
LIN {X 0,Y 346.924,Z 775.821,A -85,B 0,C 180,E1 13557.066,E2 13557.066} C_VEL
LIN {X 0,Y 339.957,Z 800.66,A -85,B 0,C 180,E1 13562.614,E2 13562.614} C_VEL
LIN {X 0,Y 335.089,Z 821.054,A -85,B 0,C 180,E1 13568.886,E2 13568.886} C_VEL
LIN {X 0,Y 332.547,Z 836.103,A -85,B 0,C 180,E1 13575.55,E2 13575.55} C_VEL
LIN {X 0,Y 331.841,Z 843.957,A -85,B 0,C 180,E1 13580.844,E2 13580.844} C_VEL
LIN {X 0,Y 331.696,Z 848.781,A -85,B 0,C 180,E1 13587.394,E2 13587.394} C_VEL
LIN {X 0,Y 331.714,Z 848.84,A -85,B 0,C 180,E1 13592.609,E2 13592.609} C_VEL
LIN {X 0,Y 331.797,Z 844.176,A -85,B 0,C 180,E1 13599.161,E2 13599.161} C_VEL
LIN {X 0,Y 332.845,Z 834.003,A -85,B 0,C 180,E1 13605.787,E2 13605.787} C_VEL
LIN {X 0,Y 335.727,Z 818.483,A -85,B 0,C 180,E1 13612.224,E2 13612.224} C_VEL
LIN {X 0,Y 341.243,Z 796.557,A -85,B 0,C 180,E1 13618.555,E2 13618.555} C_VEL
LIN {X 0,Y 344.265,Z 785.616,A -85,B 0,C 180,E1 13621.041,E2 13621.041} C_VEL
LIN {X 0,Y 343.689,Z 775.273,A -85,B 0,C 180,E1 13623.395,E2 13623.395} C_VEL
LIN {X 0,Y 343.307,Z 764.309,A -85,B 0,C 180,E1 13625.683,E2 13625.683} C_VEL
LIN {X 0,Y 352.7,Z 732.004,A -85,B 0,C 180,E1 13630.327,E2 13630.327} C_VEL
LIN {X 0,Y 361.799,Z 696.846,A -85,B 0,C 180,E1 13633.903,E2 13633.903} C_VEL
LIN {X 0,Y 369.439,Z 660.65,A -85,B 0,C 180,E1 13636.439,E2 13636.439} C_VEL
LIN {X 0,Y 371.845,Z 643.976,A -85,B 0,C 180,E1 13637.36,E2 13637.36} C_VEL
LIN {X 0,Y 358.437,Z 611.627,A -85,B 0,C 180,E1 13641.309,E2 13641.309} C_VEL
LIN {X 0,Y 340.38,Z 579.53,A -85,B 0,C 180,E1 13645.852,E2 13645.852} C_VEL
LIN {X 0,Y 323.904,Z 555.005,A -85,B 0,C 180,E1 13650.333,E2 13650.333} C_VEL
LIN {X 0,Y 321.651,Z 549.53,A -85,B 0,C 180,E1 13651.163,E2 13651.163} C_VEL
LIN {X 0,Y 322.01,Z 549.53,A -85,B 0,C 180,E1 13657.963,E2 13657.963} C_VEL
LIN {X 0,Y 322.358,Z 549.53,A -85,B 0,C 180,E1 13666.444,E2 13666.444} C_VEL
LIN {X 0,Y 323.001,Z 549.53,A -85,B 0,C 180,E1 13674.618,E2 13674.618} C_VEL
LIN {X 0,Y 323.393,Z 549.53,A -85,B 0,C 180,E1 13679.978,E2 13679.978} C_VEL
LIN {X 0,Y 322.824,Z 549.53,A -85,B 0,C 180,E1 13688.037,E2 13688.037} C_VEL
LIN {X 0,Y 322.368,Z 549.53,A -85,B 0,C 180,E1 13696.284,E2 13696.284} C_VEL
LIN {X 0,Y 322.015,Z 549.53,A -85,B 0,C 180,E1 13701.988,E2 13701.988} C_VEL
LIN {X 0,Y 321.785,Z 549.53,A -85,B 0,C 180,E1 13707.934,E2 13707.934} C_VEL
LIN {X 0,Y 321.644,Z 549.53,A -85,B 0,C 180,E1 13714.226,E2 13714.226} C_VEL
LIN {X 0,Y 321.39,Z 549.53,A -85,B 0,C 180,E1 13721.299,E2 13721.299} C_VEL
LIN {X 0,Y 321.39,Z 549.53,A -85,B 0,C 180,E1 13728.9,E2 13728.9} C_VEL
LIN {X 0,Y 321.645,Z 549.53,A -85,B 0,C 180,E1 13735.735,E2 13735.735} C_VEL
LIN {X 0,Y 321.776,Z 549.53,A -85,B 0,C 180,E1 13741.535,E2 13741.535} C_VEL
LIN {X 0,Y 323.813,Z 554.77,A -85,B 0,C 180,E1 13742.23,E2 13742.23} C_VEL
LIN {X 0,Y 334.313,Z 570.138,A -85,B 0,C 180,E1 13745.16,E2 13745.16} C_VEL
LIN {X 0,Y 349.592,Z 597.627,A -85,B 0,C 180,E1 13749.559,E2 13749.559} C_VEL
LIN {X 0,Y 361.279,Z 627.439,A -85,B 0,C 180,E1 13753.761,E2 13753.761} C_VEL
LIN {X 0,Y 363.752,Z 638.677,A -85,B 0,C 180,E1 13755.173,E2 13755.173} C_VEL
LIN {X 0,Y 356.227,Z 673.379,A -85,B 0,C 180,E1 13758.188,E2 13758.188} C_VEL
LIN {X 0,Y 348.165,Z 703.4,A -85,B 0,C 180,E1 13761.9,E2 13761.9} C_VEL
LIN {X 0,Y 340.134,Z 730.484,A -85,B 0,C 180,E1 13766.594,E2 13766.594} C_VEL
LIN {X 0,Y 332.988,Z 753.68,A -85,B 0,C 180,E1 13772.271,E2 13772.271} C_VEL
LIN {X 0,Y 328.084,Z 770.977,A -85,B 0,C 180,E1 13778.46,E2 13778.46} C_VEL
LIN {X 0,Y 325.336,Z 782.464,A -85,B 0,C 180,E1 13784.777,E2 13784.777} C_VEL
LIN {X 0,Y 324.296,Z 787.234,A -85,B 0,C 180,E1 13789.007,E2 13789.007} C_VEL
LIN {X 0,Y 323.354,Z 790.285,A -85,B 0,C 180,E1 13794.833,E2 13794.833} C_VEL
LIN {X 0,Y 323.849,Z 789.236,A -85,B 0,C 180,E1 13800.832,E2 13800.832} C_VEL
LIN {X 0,Y 325.483,Z 783.622,A -85,B 0,C 180,E1 13807.062,E2 13807.062} C_VEL
LIN {X 0,Y 328.435,Z 772.514,A -85,B 0,C 180,E1 13813.563,E2 13813.563} C_VEL
LIN {X 0,Y 333.444,Z 756.533,A -85,B 0,C 180,E1 13819.575,E2 13819.575} C_VEL
LIN {X 0,Y 341.029,Z 733.9,A -85,B 0,C 180,E1 13825.407,E2 13825.407} C_VEL
LIN {X 0,Y 349.561,Z 707.827,A -85,B 0,C 180,E1 13830.109,E2 13830.109} C_VEL
LIN {X 0,Y 358.313,Z 677.873,A -85,B 0,C 180,E1 13833.968,E2 13833.968} C_VEL
LIN {X 0,Y 366.585,Z 643.658,A -85,B 0,C 180,E1 13837.053,E2 13837.053} C_VEL
LIN {X 0,Y 366.82,Z 638.89,A -85,B 0,C 180,E1 13837.508,E2 13837.508} C_VEL
LIN {X 0,Y 358.544,Z 611.606,A -85,B 0,C 180,E1 13841.625,E2 13841.625} C_VEL
LIN {X 0,Y 347.22,Z 587.44,A -85,B 0,C 180,E1 13846,E2 13846} C_VEL
LIN {X 0,Y 336.005,Z 569.437,A -85,B 0,C 180,E1 13850.305,E2 13850.305} C_VEL
LIN {X 0,Y 331.443,Z 562.876,A -85,B 0,C 180,E1 13852.256,E2 13852.256} C_VEL
LIN {X 0,Y 327.41,Z 556.609,A -85,B 0,C 180,E1 13854.237,E2 13854.237} C_VEL
LIN {X 0,Y 323.533,Z 552.073,A -85,B 0,C 180,E1 13856.346,E2 13856.346} C_VEL
LIN {X 0,Y 323.198,Z 549.53,A -85,B 0,C 180,E1 13856.845,E2 13856.845} C_VEL
LIN {X 0,Y 323.208,Z 549.53,A -85,B 0,C 180,E1 13862.698,E2 13862.698} C_VEL
LIN {X 0,Y 322.671,Z 549.53,A -85,B 0,C 180,E1 13870.871,E2 13870.871} C_VEL
LIN {X 0,Y 322.367,Z 549.53,A -85,B 0,C 180,E1 13876.331,E2 13876.331} C_VEL
LIN {X 0,Y 322.01,Z 549.872,A -85,B 0,C 180,E1 13882.898,E2 13882.898} C_VEL
LIN {X 0,Y 324.184,Z 555.02,A -85,B 0,C 180,E1 13884.385,E2 13884.385} C_VEL
LIN {X 0,Y 327.574,Z 558.162,A -85,B 0,C 180,E1 13886.123,E2 13886.123} C_VEL
LIN {X 0,Y 331.651,Z 563.758,A -85,B 0,C 180,E1 13888.052,E2 13888.052} C_VEL
LIN {X 0,Y 345.346,Z 583.659,A -85,B 0,C 180,E1 13893.232,E2 13893.232} C_VEL
LIN {X 0,Y 359.138,Z 608.16,A -85,B 0,C 180,E1 13897.619,E2 13897.619} C_VEL
LIN {X 0,Y 371.203,Z 637.724,A -85,B 0,C 180,E1 13901.674,E2 13901.674} C_VEL
LIN {X 0,Y 373.039,Z 646.678,A -85,B 0,C 180,E1 13902.636,E2 13902.636} C_VEL
LIN {X 0,Y 365.619,Z 683.576,A -85,B 0,C 180,E1 13904.906,E2 13904.906} C_VEL
LIN {X 0,Y 356.417,Z 719.702,A -85,B 0,C 180,E1 13908.18,E2 13908.18} C_VEL
LIN {X 0,Y 346.358,Z 754.217,A -85,B 0,C 180,E1 13912.68,E2 13912.68} C_VEL
LIN {X 0,Y 338.102,Z 781.542,A -85,B 0,C 180,E1 13917.619,E2 13917.619} C_VEL
LIN {X 0,Y 331.052,Z 805.85,A -85,B 0,C 180,E1 13923.615,E2 13923.615} C_VEL
LIN {X 0,Y 326.693,Z 823.837,A -85,B 0,C 180,E1 13929.733,E2 13929.733} C_VEL
LIN {X 0,Y 324.43,Z 837.666,A -85,B 0,C 180,E1 13936.554,E2 13936.554} C_VEL
LIN {X 0,Y 323.859,Z 844.571,A -85,B 0,C 180,E1 13941.967,E2 13941.967} C_VEL
LIN {X 0,Y 323.811,Z 848.074,A -85,B 0,C 180,E1 13947.331,E2 13947.331} C_VEL
LIN {X 0,Y 323.83,Z 848.129,A -85,B 0,C 180,E1 13952.673,E2 13952.673} C_VEL
LIN {X 0,Y 323.917,Z 843.445,A -85,B 0,C 180,E1 13959.386,E2 13959.386} C_VEL
LIN {X 0,Y 325.07,Z 833.246,A -85,B 0,C 180,E1 13966.174,E2 13966.174} C_VEL
LIN {X 0,Y 328.524,Z 816.239,A -85,B 0,C 180,E1 13973.245,E2 13973.245} C_VEL
LIN {X 0,Y 334.109,Z 795.301,A -85,B 0,C 180,E1 13979.32,E2 13979.32} C_VEL
LIN {X 0,Y 341.555,Z 770.039,A -85,B 0,C 180,E1 13984.671,E2 13984.671} C_VEL
LIN {X 0,Y 343.307,Z 764.309,A -85,B 0,C 180,E1 13985.683,E2 13985.683} C_VEL
LIN {X 0,Y 343.282,Z 752.768,A -85,B 0,C 180,E1 13987.896,E2 13987.896} C_VEL
LIN {X 0,Y 343.593,Z 740.455,A -85,B 0,C 180,E1 13989.973,E2 13989.973} C_VEL
LIN {X 0,Y 353.095,Z 706.862,A -85,B 0,C 180,E1 13993.775,E2 13993.775} C_VEL
LIN {X 0,Y 361.291,Z 671.891,A -85,B 0,C 180,E1 13996.563,E2 13996.563} C_VEL
LIN {X 0,Y 365.484,Z 646.357,A -85,B 0,C 180,E1 13998.098,E2 13998.098} C_VEL
LIN {X 0,Y 351.49,Z 612.348,A -85,B 0,C 180,E1 14002.46,E2 14002.46} C_VEL
LIN {X 0,Y 334.876,Z 583.068,A -85,B 0,C 180,E1 14006.865,E2 14006.865} C_VEL
LIN {X 0,Y 316.692,Z 555.665,A -85,B 0,C 180,E1 14012.106,E2 14012.106} C_VEL
LIN {X 0,Y 313.993,Z 551.009,A -85,B 0,C 180,E1 14013.01,E2 14013.01} C_VEL
LIN {X 0,Y 313.838,Z 549.53,A -85,B 0,C 180,E1 14013.317,E2 14013.317} C_VEL
LIN {X 0,Y 314.147,Z 549.53,A -85,B 0,C 180,E1 14020.332,E2 14020.332} C_VEL
LIN {X 0,Y 314.4,Z 549.53,A -85,B 0,C 180,E1 14026.094,E2 14026.094} C_VEL
LIN {X 0,Y 315.08,Z 549.53,A -85,B 0,C 180,E1 14034.482,E2 14034.482} C_VEL
LIN {X 0,Y 315.493,Z 549.53,A -85,B 0,C 180,E1 14039.977,E2 14039.977} C_VEL
LIN {X 0,Y 314.905,Z 549.53,A -85,B 0,C 180,E1 14048.24,E2 14048.24} C_VEL
LIN {X 0,Y 314.414,Z 549.53,A -85,B 0,C 180,E1 14056.708,E2 14056.708} C_VEL
LIN {X 0,Y 313.915,Z 549.53,A -85,B 0,C 180,E1 14065.603,E2 14065.603} C_VEL
LIN {X 0,Y 313.728,Z 549.53,A -85,B 0,C 180,E1 14071.909,E2 14071.909} C_VEL
LIN {X 0,Y 313.43,Z 549.53,A -85,B 0,C 180,E1 14079.614,E2 14079.614} C_VEL
LIN {X 0,Y 313.354,Z 549.53,A -85,B 0,C 180,E1 14087.606,E2 14087.606} C_VEL
LIN {X 0,Y 313.648,Z 549.53,A -85,B 0,C 180,E1 14094.816,E2 14094.816} C_VEL
LIN {X 0,Y 313.807,Z 550.094,A -85,B 0,C 180,E1 14099.557,E2 14099.557} C_VEL
LIN {X 0,Y 316.399,Z 555.332,A -85,B 0,C 180,E1 14100.444,E2 14100.444} C_VEL
LIN {X 0,Y 330.818,Z 576.983,A -85,B 0,C 180,E1 14104.737,E2 14104.737} C_VEL
LIN {X 0,Y 345.257,Z 604.249,A -85,B 0,C 180,E1 14109.261,E2 14109.261} C_VEL
LIN {X 0,Y 355.519,Z 632.003,A -85,B 0,C 180,E1 14113.297,E2 14113.297} C_VEL
LIN {X 0,Y 357.291,Z 641.727,A -85,B 0,C 180,E1 14114.53,E2 14114.53} C_VEL
LIN {X 0,Y 349.653,Z 675.181,A -85,B 0,C 180,E1 14117.536,E2 14117.536} C_VEL
LIN {X 0,Y 341.137,Z 705.619,A -85,B 0,C 180,E1 14121.412,E2 14121.412} C_VEL
LIN {X 0,Y 332.755,Z 732.586,A -85,B 0,C 180,E1 14126.239,E2 14126.239} C_VEL
LIN {X 0,Y 325.404,Z 755.192,A -85,B 0,C 180,E1 14131.991,E2 14131.991} C_VEL
LIN {X 0,Y 320.439,Z 771.808,A -85,B 0,C 180,E1 14138.12,E2 14138.12} C_VEL
LIN {X 0,Y 317.79,Z 782.072,A -85,B 0,C 180,E1 14143.732,E2 14143.732} C_VEL
LIN {X 0,Y 316.3,Z 788.513,A -85,B 0,C 180,E1 14149.507,E2 14149.507} C_VEL
LIN {X 0,Y 315.443,Z 791.103,A -85,B 0,C 180,E1 14155.5,E2 14155.5} C_VEL
LIN {X 0,Y 316.169,Z 789.566,A -85,B 0,C 180,E1 14161.666,E2 14161.666} C_VEL
LIN {X 0,Y 317.946,Z 783.416,A -85,B 0,C 180,E1 14168.095,E2 14168.095} C_VEL
LIN {X 0,Y 321.445,Z 771.706,A -85,B 0,C 180,E1 14174.76,E2 14174.76} C_VEL
LIN {X 0,Y 327.173,Z 754.705,A -85,B 0,C 180,E1 14180.983,E2 14180.983} C_VEL
LIN {X 0,Y 334.984,Z 732.689,A -85,B 0,C 180,E1 14186.533,E2 14186.533} C_VEL
LIN {X 0,Y 344.059,Z 705.981,A -85,B 0,C 180,E1 14191.3,E2 14191.3} C_VEL
LIN {X 0,Y 353.434,Z 675.053,A -85,B 0,C 180,E1 14195.199,E2 14195.199} C_VEL
LIN {X 0,Y 361.093,Z 642.898,A -85,B 0,C 180,E1 14198.084,E2 14198.084} C_VEL
LIN {X 0,Y 353.209,Z 615.413,A -85,B 0,C 180,E1 14202.396,E2 14202.396} C_VEL
LIN {X 0,Y 342.749,Z 592.407,A -85,B 0,C 180,E1 14206.824,E2 14206.824} C_VEL
LIN {X 0,Y 332.702,Z 575.545,A -85,B 0,C 180,E1 14211.054,E2 14211.054} C_VEL
LIN {X 0,Y 324.952,Z 563.727,A -85,B 0,C 180,E1 14214.861,E2 14214.861} C_VEL
LIN {X 0,Y 321.126,Z 558.037,A -85,B 0,C 180,E1 14217.161,E2 14217.161} C_VEL
LIN {X 0,Y 315.491,Z 551.18,A -85,B 0,C 180,E1 14221.563,E2 14221.563} C_VEL
LIN {X 0,Y 315.302,Z 549.53,A -85,B 0,C 180,E1 14222.079,E2 14222.079} C_VEL
LIN {X 0,Y 314.904,Z 549.53,A -85,B 0,C 180,E1 14228.287,E2 14228.287} C_VEL
LIN {X 0,Y 314.481,Z 549.53,A -85,B 0,C 180,E1 14236.332,E2 14236.332} C_VEL
LIN {X 0,Y 314.337,Z 550.367,A -85,B 0,C 180,E1 14237.48,E2 14237.48} C_VEL
LIN {X 0,Y 317.025,Z 555.585,A -85,B 0,C 180,E1 14240.287,E2 14240.287} C_VEL
LIN {X 0,Y 320.205,Z 558.311,A -85,B 0,C 180,E1 14242.532,E2 14242.532} C_VEL
LIN {X 0,Y 324.24,Z 563.989,A -85,B 0,C 180,E1 14245.005,E2 14245.005} C_VEL
LIN {X 0,Y 331.499,Z 574.561,A -85,B 0,C 180,E1 14248.555,E2 14248.555} C_VEL
LIN {X 0,Y 342.259,Z 590.312,A -85,B 0,C 180,E1 14252.705,E2 14252.705} C_VEL
LIN {X 0,Y 354.812,Z 613.637,A -85,B 0,C 180,E1 14257.033,E2 14257.033} C_VEL
LIN {X 0,Y 365.806,Z 642.26,A -85,B 0,C 180,E1 14261.119,E2 14261.119} C_VEL
LIN {X 0,Y 367.155,Z 648.781,A -85,B 0,C 180,E1 14261.849,E2 14261.849} C_VEL
LIN {X 0,Y 358.872,Z 687.702,A -85,B 0,C 180,E1 14264.373,E2 14264.373} C_VEL
LIN {X 0,Y 349.239,Z 722.866,A -85,B 0,C 180,E1 14267.731,E2 14267.731} C_VEL
LIN {X 0,Y 339.631,Z 754.126,A -85,B 0,C 180,E1 14271.943,E2 14271.943} C_VEL
LIN {X 0,Y 330.542,Z 782.694,A -85,B 0,C 180,E1 14277.269,E2 14277.269} C_VEL
LIN {X 0,Y 323.361,Z 806.25,A -85,B 0,C 180,E1 14283.312,E2 14283.312} C_VEL
LIN {X 0,Y 318.651,Z 824.728,A -85,B 0,C 180,E1 14289.922,E2 14289.922} C_VEL
LIN {X 0,Y 316.592,Z 836.942,A -85,B 0,C 180,E1 14296.215,E2 14296.215} C_VEL
LIN {X 0,Y 315.981,Z 843.854,A -85,B 0,C 180,E1 14301.765,E2 14301.765} C_VEL
LIN {X 0,Y 315.947,Z 847.37,A -85,B 0,C 180,E1 14307.264,E2 14307.264} C_VEL
LIN {X 0,Y 315.962,Z 847.418,A -85,B 0,C 180,E1 14312.739,E2 14312.739} C_VEL
LIN {X 0,Y 316.044,Z 842.713,A -85,B 0,C 180,E1 14319.622,E2 14319.622} C_VEL
LIN {X 0,Y 317.289,Z 832.477,A -85,B 0,C 180,E1 14326.582,E2 14326.582} C_VEL
LIN {X 0,Y 320.709,Z 816.613,A -85,B 0,C 180,E1 14333.411,E2 14333.411} C_VEL
LIN {X 0,Y 326.653,Z 795.39,A -85,B 0,C 180,E1 14339.785,E2 14339.785} C_VEL
LIN {X 0,Y 334.81,Z 769.022,A -85,B 0,C 180,E1 14345.473,E2 14345.473} C_VEL
LIN {X 0,Y 343.593,Z 740.455,A -85,B 0,C 180,E1 14349.973,E2 14349.973} C_VEL
LIN {X 0,Y 344.127,Z 727.627,A -85,B 0,C 180,E1 14351.959,E2 14351.959} C_VEL
LIN {X 0,Y 344.336,Z 716.03,A -85,B 0,C 180,E1 14353.644,E2 14353.644} C_VEL
LIN {X 0,Y 344.774,Z 714.217,A -85,B 0,C 180,E1 14353.844,E2 14353.844} C_VEL
LIN {X 0,Y 353.825,Z 678.552,A -85,B 0,C 180,E1 14356.955,E2 14356.955} C_VEL
LIN {X 0,Y 359.43,Z 649.807,A -85,B 0,C 180,E1 14358.742,E2 14358.742} C_VEL
LIN {X 0,Y 346.154,Z 616.495,A -85,B 0,C 180,E1 14363.168,E2 14363.168} C_VEL
LIN {X 0,Y 329.481,Z 586.264,A -85,B 0,C 180,E1 14367.91,E2 14367.91} C_VEL
LIN {X 0,Y 312.654,Z 561.342,A -85,B 0,C 180,E1 14372.945,E2 14372.945} C_VEL
LIN {X 0,Y 308.902,Z 555.704,A -85,B 0,C 180,E1 14374.214,E2 14374.214} C_VEL
LIN {X 0,Y 306.092,Z 551.045,A -85,B 0,C 180,E1 14375.228,E2 14375.228} C_VEL
LIN {X 0,Y 305.95,Z 549.53,A -85,B 0,C 180,E1 14375.499,E2 14375.499} C_VEL
LIN {X 0,Y 306.316,Z 549.53,A -85,B 0,C 180,E1 14382.787,E2 14382.787} C_VEL
LIN {X 0,Y 306.896,Z 549.53,A -85,B 0,C 180,E1 14391.496,E2 14391.496} C_VEL
LIN {X 0,Y 307.465,Z 549.53,A -85,B 0,C 180,E1 14397.164,E2 14397.164} C_VEL
LIN {X 0,Y 307.413,Z 549.53,A -85,B 0,C 180,E1 14402.79,E2 14402.79} C_VEL
LIN {X 0,Y 306.821,Z 549.53,A -85,B 0,C 180,E1 14411.319,E2 14411.319} C_VEL
LIN {X 0,Y 306.428,Z 549.53,A -85,B 0,C 180,E1 14417.157,E2 14417.157} C_VEL
LIN {X 0,Y 306.07,Z 549.53,A -85,B 0,C 180,E1 14423.199,E2 14423.199} C_VEL
LIN {X 0,Y 305.813,Z 549.53,A -85,B 0,C 180,E1 14429.532,E2 14429.532} C_VEL
LIN {X 0,Y 305.544,Z 549.53,A -85,B 0,C 180,E1 14437.792,E2 14437.792} C_VEL
LIN {X 0,Y 305.46,Z 549.53,A -85,B 0,C 180,E1 14446.239,E2 14446.239} C_VEL
LIN {X 0,Y 305.567,Z 549.53,A -85,B 0,C 180,E1 14453.655,E2 14453.655} C_VEL
LIN {X 0,Y 305.743,Z 549.817,A -85,B 0,C 180,E1 14457.319,E2 14457.319} C_VEL
LIN {X 0,Y 308.091,Z 555.077,A -85,B 0,C 180,E1 14458.22,E2 14458.22} C_VEL
LIN {X 0,Y 310.733,Z 558.353,A -85,B 0,C 180,E1 14459.092,E2 14459.092} C_VEL
LIN {X 0,Y 326.409,Z 582.337,A -85,B 0,C 180,E1 14464.077,E2 14464.077} C_VEL
LIN {X 0,Y 340.021,Z 609.006,A -85,B 0,C 180,E1 14468.653,E2 14468.653} C_VEL
LIN {X 0,Y 349.797,Z 636.872,A -85,B 0,C 180,E1 14472.882,E2 14472.882} C_VEL
LIN {X 0,Y 351.026,Z 643.923,A -85,B 0,C 180,E1 14473.815,E2 14473.815} C_VEL
LIN {X 0,Y 342.849,Z 677.937,A -85,B 0,C 180,E1 14476.962,E2 14476.962} C_VEL
LIN {X 0,Y 334.087,Z 707.859,A -85,B 0,C 180,E1 14480.902,E2 14480.902} C_VEL
LIN {X 0,Y 325.248,Z 734.865,A -85,B 0,C 180,E1 14485.921,E2 14485.921} C_VEL
LIN {X 0,Y 317.802,Z 756.766,A -85,B 0,C 180,E1 14491.719,E2 14491.719} C_VEL
LIN {X 0,Y 312.93,Z 772.316,A -85,B 0,C 180,E1 14497.618,E2 14497.618} C_VEL
LIN {X 0,Y 309.806,Z 783.638,A -85,B 0,C 180,E1 14504.094,E2 14504.094} C_VEL
LIN {X 0,Y 308.27,Z 789.66,A -85,B 0,C 180,E1 14510.037,E2 14510.037} C_VEL
LIN {X 0,Y 307.553,Z 791.895,A -85,B 0,C 180,E1 14516.203,E2 14516.203} C_VEL
LIN {X 0,Y 308.537,Z 789.898,A -85,B 0,C 180,E1 14522.545,E2 14522.545} C_VEL
LIN {X 0,Y 310.511,Z 783.216,A -85,B 0,C 180,E1 14529.178,E2 14529.178} C_VEL
LIN {X 0,Y 314.514,Z 770.755,A -85,B 0,C 180,E1 14536.026,E2 14536.026} C_VEL
LIN {X 0,Y 320.967,Z 753.008,A -85,B 0,C 180,E1 14542.363,E2 14542.363} C_VEL
LIN {X 0,Y 329.513,Z 730.394,A -85,B 0,C 180,E1 14547.93,E2 14547.93} C_VEL
LIN {X 0,Y 339.362,Z 702.336,A -85,B 0,C 180,E1 14552.784,E2 14552.784} C_VEL
LIN {X 0,Y 349.027,Z 670.907,A -85,B 0,C 180,E1 14556.572,E2 14556.572} C_VEL
LIN {X 0,Y 355.104,Z 645.675,A -85,B 0,C 180,E1 14558.854,E2 14558.854} C_VEL
LIN {X 0,Y 347.796,Z 618.952,A -85,B 0,C 180,E1 14563.258,E2 14563.258} C_VEL
LIN {X 0,Y 337.231,Z 594.856,A -85,B 0,C 180,E1 14568.178,E2 14568.178} C_VEL
LIN {X 0,Y 326.811,Z 577.183,A -85,B 0,C 180,E1 14573.139,E2 14573.139} C_VEL
LIN {X 0,Y 322.231,Z 570.495,A -85,B 0,C 180,E1 14575.659,E2 14575.659} C_VEL
LIN {X 0,Y 318.012,Z 564.142,A -85,B 0,C 180,E1 14578.443,E2 14578.443} C_VEL
LIN {X 0,Y 313.813,Z 558.128,A -85,B 0,C 180,E1 14582.175,E2 14582.175} C_VEL
LIN {X 0,Y 310.097,Z 555.818,A -85,B 0,C 180,E1 14588.416,E2 14588.416} C_VEL
LIN {X 0,Y 312.86,Z 557.924,A -85,B 0,C 180,E1 14597.022,E2 14597.022} C_VEL
LIN {X 0,Y 316.153,Z 563.669,A -85,B 0,C 180,E1 14600.447,E2 14600.447} C_VEL
LIN {X 0,Y 318.442,Z 565.925,A -85,B 0,C 180,E1 14602.114,E2 14602.114} C_VEL
LIN {X 0,Y 324.169,Z 574.365,A -85,B 0,C 180,E1 14605.628,E2 14605.628} C_VEL
LIN {X 0,Y 332.613,Z 586.631,A -85,B 0,C 180,E1 14609.586,E2 14609.586} C_VEL
LIN {X 0,Y 344.444,Z 606.412,A -85,B 0,C 180,E1 14614.176,E2 14614.176} C_VEL
LIN {X 0,Y 356.384,Z 634.068,A -85,B 0,C 180,E1 14618.761,E2 14618.761} C_VEL
LIN {X 0,Y 361.357,Z 650.801,A -85,B 0,C 180,E1 14621.04,E2 14621.04} C_VEL
LIN {X 0,Y 353.229,Z 687.035,A -85,B 0,C 180,E1 14623.43,E2 14623.43} C_VEL
LIN {X 0,Y 343.213,Z 722.32,A -85,B 0,C 180,E1 14626.832,E2 14626.832} C_VEL
LIN {X 0,Y 333.169,Z 753.419,A -85,B 0,C 180,E1 14631.068,E2 14631.068} C_VEL
LIN {X 0,Y 323.644,Z 781.877,A -85,B 0,C 180,E1 14636.459,E2 14636.459} C_VEL
LIN {X 0,Y 315.989,Z 805.505,A -85,B 0,C 180,E1 14642.638,E2 14642.638} C_VEL
LIN {X 0,Y 311.023,Z 824.004,A -85,B 0,C 180,E1 14649.408,E2 14649.408} C_VEL
LIN {X 0,Y 308.764,Z 836.218,A -85,B 0,C 180,E1 14655.858,E2 14655.858} C_VEL
LIN {X 0,Y 308.102,Z 843.144,A -85,B 0,C 180,E1 14661.553,E2 14661.553} C_VEL
LIN {X 0,Y 308.061,Z 846.664,A -85,B 0,C 180,E1 14667.194,E2 14667.194} C_VEL
LIN {X 0,Y 308.077,Z 846.705,A -85,B 0,C 180,E1 14672.81,E2 14672.81} C_VEL
LIN {X 0,Y 308.18,Z 841.975,A -85,B 0,C 180,E1 14679.87,E2 14679.87} C_VEL
LIN {X 0,Y 309.528,Z 831.697,A -85,B 0,C 180,E1 14687.011,E2 14687.011} C_VEL
LIN {X 0,Y 313.074,Z 816.133,A -85,B 0,C 180,E1 14693.886,E2 14693.886} C_VEL
LIN {X 0,Y 319.506,Z 794.485,A -85,B 0,C 180,E1 14700.514,E2 14700.514} C_VEL
LIN {X 0,Y 328.102,Z 768.034,A -85,B 0,C 180,E1 14706.305,E2 14706.305} C_VEL
LIN {X 0,Y 337.389,Z 739.094,A -85,B 0,C 180,E1 14710.891,E2 14710.891} C_VEL
LIN {X 0,Y 344.774,Z 714.217,A -85,B 0,C 180,E1 14713.844,E2 14713.844} C_VEL
LIN {X 0,Y 345.54,Z 700.354,A -85,B 0,C 180,E1 14715.629,E2 14715.629} C_VEL
LIN {X 0,Y 346.114,Z 685.881,A -85,B 0,C 180,E1 14717.261,E2 14717.261} C_VEL
LIN {X 0,Y 353.212,Z 652.602,A -85,B 0,C 180,E1 14719.466,E2 14719.466} C_VEL
LIN {X 0,Y 340.764,Z 620.536,A -85,B 0,C 180,E1 14723.916,E2 14723.916} C_VEL
LIN {X 0,Y 325.256,Z 591.796,A -85,B 0,C 180,E1 14728.617,E2 14728.617} C_VEL
LIN {X 0,Y 309.132,Z 567.344,A -85,B 0,C 180,E1 14733.655,E2 14733.655} C_VEL
LIN {X 0,Y 301.079,Z 555.685,A -85,B 0,C 180,E1 14736.537,E2 14736.537} C_VEL
LIN {X 0,Y 298.215,Z 550.862,A -85,B 0,C 180,E1 14737.676,E2 14737.676} C_VEL
LIN {X 0,Y 298.118,Z 549.53,A -85,B 0,C 180,E1 14738.06,E2 14738.06} C_VEL
LIN {X 0,Y 298.512,Z 549.53,A -85,B 0,C 180,E1 14745.338,E2 14745.338} C_VEL
LIN {X 0,Y 299.209,Z 549.53,A -85,B 0,C 180,E1 14754.188,E2 14754.188} C_VEL
LIN {X 0,Y 299.694,Z 549.53,A -85,B 0,C 180,E1 14759.976,E2 14759.976} C_VEL
LIN {X 0,Y 299.038,Z 549.53,A -85,B 0,C 180,E1 14768.681,E2 14768.681} C_VEL
LIN {X 0,Y 298.523,Z 549.53,A -85,B 0,C 180,E1 14776.163,E2 14776.163} C_VEL
LIN {X 0,Y 298.006,Z 549.53,A -85,B 0,C 180,E1 14784.286,E2 14784.286} C_VEL
LIN {X 0,Y 297.78,Z 549.53,A -85,B 0,C 180,E1 14790.512,E2 14790.512} C_VEL
LIN {X 0,Y 297.633,Z 549.53,A -85,B 0,C 180,E1 14797.434,E2 14797.434} C_VEL
LIN {X 0,Y 297.495,Z 549.53,A -85,B 0,C 180,E1 14805.198,E2 14805.198} C_VEL
LIN {X 0,Y 297.624,Z 549.53,A -85,B 0,C 180,E1 14812.522,E2 14812.522} C_VEL
LIN {X 0,Y 297.629,Z 550.214,A -85,B 0,C 180,E1 14814.859,E2 14814.859} C_VEL
LIN {X 0,Y 300.15,Z 555.312,A -85,B 0,C 180,E1 14815.904,E2 14815.904} C_VEL
LIN {X 0,Y 302.88,Z 558.404,A -85,B 0,C 180,E1 14816.88,E2 14816.88} C_VEL
LIN {X 0,Y 318.333,Z 581.385,A -85,B 0,C 180,E1 14822.168,E2 14822.168} C_VEL
LIN {X 0,Y 332.455,Z 608.453,A -85,B 0,C 180,E1 14827.16,E2 14827.16} C_VEL
LIN {X 0,Y 342.25,Z 635.182,A -85,B 0,C 180,E1 14831.457,E2 14831.457} C_VEL
LIN {X 0,Y 344.718,Z 646.344,A -85,B 0,C 180,E1 14833.089,E2 14833.089} C_VEL
LIN {X 0,Y 336.081,Z 680.646,A -85,B 0,C 180,E1 14836.364,E2 14836.364} C_VEL
LIN {X 0,Y 326.472,Z 711.957,A -85,B 0,C 180,E1 14840.688,E2 14840.688} C_VEL
LIN {X 0,Y 317.584,Z 737.57,A -85,B 0,C 180,E1 14845.705,E2 14845.705} C_VEL
LIN {X 0,Y 309.955,Z 759.074,A -85,B 0,C 180,E1 14851.679,E2 14851.679} C_VEL
LIN {X 0,Y 304.462,Z 775.846,A -85,B 0,C 180,E1 14858.549,E2 14858.549} C_VEL
LIN {X 0,Y 301.855,Z 785.2,A -85,B 0,C 180,E1 14864.473,E2 14864.473} C_VEL
LIN {X 0,Y 300.271,Z 790.783,A -85,B 0,C 180,E1 14870.594,E2 14870.594} C_VEL
LIN {X 0,Y 299.716,Z 792.551,A -85,B 0,C 180,E1 14876.942,E2 14876.942} C_VEL
LIN {X 0,Y 300.875,Z 790.105,A -85,B 0,C 180,E1 14883.481,E2 14883.481} C_VEL
LIN {X 0,Y 303.157,Z 782.85,A -85,B 0,C 180,E1 14890.32,E2 14890.32} C_VEL
LIN {X 0,Y 307.769,Z 769.756,A -85,B 0,C 180,E1 14897.343,E2 14897.343} C_VEL
LIN {X 0,Y 314.978,Z 751.307,A -85,B 0,C 180,E1 14903.799,E2 14903.799} C_VEL
LIN {X 0,Y 324.468,Z 727.241,A -85,B 0,C 180,E1 14909.531,E2 14909.531} C_VEL
LIN {X 0,Y 334.418,Z 699.839,A -85,B 0,C 180,E1 14914.121,E2 14914.121} C_VEL
LIN {X 0,Y 344.419,Z 668.106,A -85,B 0,C 180,E1 14917.849,E2 14917.849} C_VEL
LIN {X 0,Y 349.209,Z 648.693,A -85,B 0,C 180,E1 14919.614,E2 14919.614} C_VEL
LIN {X 0,Y 342.648,Z 622.934,A -85,B 0,C 180,E1 14924.069,E2 14924.069} C_VEL
LIN {X 0,Y 333.182,Z 600.396,A -85,B 0,C 180,E1 14928.927,E2 14928.927} C_VEL
LIN {X 0,Y 324.03,Z 583.859,A -85,B 0,C 180,E1 14933.746,E2 14933.746} C_VEL
LIN {X 0,Y 319.54,Z 577.047,A -85,B 0,C 180,E1 14936.449,E2 14936.449} C_VEL
LIN {X 0,Y 316.151,Z 571.522,A -85,B 0,C 180,E1 14938.953,E2 14938.953} C_VEL
LIN {X 0,Y 311.601,Z 564.802,A -85,B 0,C 180,E1 14943.493,E2 14943.493} C_VEL
LIN {X 0,Y 309.235,Z 563.956,A -85,B 0,C 180,E1 14952.597,E2 14952.597} C_VEL
LIN {X 0,Y 311.527,Z 565.889,A -85,B 0,C 180,E1 14956.735,E2 14956.735} C_VEL
LIN {X 0,Y 315.613,Z 571.911,A -85,B 0,C 180,E1 14960.85,E2 14960.85} C_VEL
LIN {X 0,Y 322.265,Z 581.885,A -85,B 0,C 180,E1 14965.26,E2 14965.26} C_VEL
LIN {X 0,Y 330.505,Z 594.376,A -85,B 0,C 180,E1 14969.318,E2 14969.318} C_VEL
LIN {X 0,Y 341.037,Z 613.39,A -85,B 0,C 180,E1 14973.787,E2 14973.787} C_VEL
LIN {X 0,Y 351.733,Z 640.11,A -85,B 0,C 180,E1 14978.34,E2 14978.34} C_VEL
LIN {X 0,Y 355.399,Z 653.831,A -85,B 0,C 180,E1 14980.268,E2 14980.268} C_VEL
LIN {X 0,Y 346.827,Z 689.918,A -85,B 0,C 180,E1 14982.762,E2 14982.762} C_VEL
LIN {X 0,Y 336.709,Z 723.559,A -85,B 0,C 180,E1 14986.111,E2 14986.111} C_VEL
LIN {X 0,Y 326.124,Z 754.702,A -85,B 0,C 180,E1 14990.491,E2 14990.491} C_VEL
LIN {X 0,Y 316.312,Z 782.569,A -85,B 0,C 180,E1 14995.954,E2 14995.954} C_VEL
LIN {X 0,Y 308.551,Z 805.174,A -85,B 0,C 180,E1 15002.055,E2 15002.055} C_VEL
LIN {X 0,Y 303.397,Z 823.28,A -85,B 0,C 180,E1 15008.866,E2 15008.866} C_VEL
LIN {X 0,Y 300.81,Z 836.548,A -85,B 0,C 180,E1 15016.217,E2 15016.217} C_VEL
LIN {X 0,Y 300.154,Z 843.648,A -85,B 0,C 180,E1 15022.782,E2 15022.782} C_VEL
LIN {X 0,Y 300.475,Z 846.448,A -85,B 0,C 180,E1 15030.002,E2 15030.002} C_VEL
LIN {X 0,Y 300.152,Z 843.8,A -85,B 0,C 180,E1 15037.223,E2 15037.223} C_VEL
LIN {X 0,Y 300.955,Z 835.723,A -85,B 0,C 180,E1 15044.521,E2 15044.521} C_VEL
LIN {X 0,Y 303.787,Z 821.848,A -85,B 0,C 180,E1 15051.875,E2 15051.875} C_VEL
LIN {X 0,Y 309.842,Z 801.25,A -85,B 0,C 180,E1 15059.148,E2 15059.148} C_VEL
LIN {X 0,Y 318.265,Z 776.308,A -85,B 0,C 180,E1 15065.327,E2 15065.327} C_VEL
LIN {X 0,Y 327.902,Z 747.789,A -85,B 0,C 180,E1 15070.412,E2 15070.412} C_VEL
LIN {X 0,Y 338.222,Z 715.127,A -85,B 0,C 180,E1 15074.565,E2 15074.565} C_VEL
LIN {X 0,Y 346.114,Z 685.881,A -85,B 0,C 180,E1 15077.261,E2 15077.261} C_VEL
LIN {X 0,Y 347.356,Z 670.743,A -85,B 0,C 180,E1 15078.693,E2 15078.693} C_VEL
LIN {X 0,Y 346.894,Z 655.607,A -85,B 0,C 180,E1 15080.2,E2 15080.2} C_VEL
LIN {X 0,Y 335.817,Z 625.506,A -85,B 0,C 180,E1 15084.536,E2 15084.536} C_VEL
LIN {X 0,Y 321.33,Z 597.568,A -85,B 0,C 180,E1 15089.271,E2 15089.271} C_VEL
LIN {X 0,Y 303.2,Z 569.391,A -85,B 0,C 180,E1 15095.265,E2 15095.265} C_VEL
LIN {X 0,Y 293.545,Z 555.936,A -85,B 0,C 180,E1 15098.995,E2 15098.995} C_VEL
LIN {X 0,Y 290.377,Z 550.882,A -85,B 0,C 180,E1 15100.377,E2 15100.377} C_VEL
LIN {X 0,Y 290.255,Z 549.53,A -85,B 0,C 180,E1 15100.656,E2 15100.656} C_VEL
LIN {X 0,Y 290.754,Z 549.53,A -85,B 0,C 180,E1 15107.996,E2 15107.996} C_VEL
LIN {X 0,Y 291.641,Z 549.53,A -85,B 0,C 180,E1 15117.01,E2 15117.01} C_VEL
LIN {X 0,Y 291.585,Z 549.53,A -85,B 0,C 180,E1 15122.941,E2 15122.941} C_VEL
LIN {X 0,Y 290.901,Z 549.53,A -85,B 0,C 180,E1 15131.947,E2 15131.947} C_VEL
LIN {X 0,Y 290.339,Z 549.53,A -85,B 0,C 180,E1 15140.679,E2 15140.679} C_VEL
LIN {X 0,Y 289.934,Z 549.53,A -85,B 0,C 180,E1 15147.897,E2 15147.897} C_VEL
LIN {X 0,Y 289.744,Z 549.53,A -85,B 0,C 180,E1 15154.912,E2 15154.912} C_VEL
LIN {X 0,Y 289.473,Z 549.53,A -85,B 0,C 180,E1 15163.126,E2 15163.126} C_VEL
LIN {X 0,Y 289.681,Z 549.53,A -85,B 0,C 180,E1 15172.062,E2 15172.062} C_VEL
LIN {X 0,Y 292.043,Z 555.126,A -85,B 0,C 180,E1 15173.249,E2 15173.249} C_VEL
LIN {X 0,Y 294.771,Z 558.207,A -85,B 0,C 180,E1 15174.335,E2 15174.335} C_VEL
LIN {X 0,Y 308.444,Z 577.926,A -85,B 0,C 180,E1 15179.44,E2 15179.44} C_VEL
LIN {X 0,Y 322.583,Z 602.886,A -85,B 0,C 180,E1 15184.652,E2 15184.652} C_VEL
LIN {X 0,Y 333.914,Z 630.836,A -85,B 0,C 180,E1 15189.515,E2 15189.515} C_VEL
LIN {X 0,Y 338.568,Z 648.507,A -85,B 0,C 180,E1 15192.322,E2 15192.322} C_VEL
LIN {X 0,Y 329.346,Z 683.338,A -85,B 0,C 180,E1 15195.741,E2 15195.741} C_VEL
LIN {X 0,Y 319.453,Z 714.02,A -85,B 0,C 180,E1 15200.138,E2 15200.138} C_VEL
LIN {X 0,Y 310.179,Z 739.543,A -85,B 0,C 180,E1 15205.305,E2 15205.305} C_VEL
LIN {X 0,Y 302.122,Z 761.308,A -85,B 0,C 180,E1 15211.612,E2 15211.612} C_VEL
LIN {X 0,Y 296.845,Z 776.567,A -85,B 0,C 180,E1 15218.142,E2 15218.142} C_VEL
LIN {X 0,Y 293.899,Z 786.69,A -85,B 0,C 180,E1 15224.873,E2 15224.873} C_VEL
LIN {X 0,Y 292.138,Z 792.175,A -85,B 0,C 180,E1 15231.701,E2 15231.701} C_VEL
LIN {X 0,Y 291.929,Z 793.136,A -85,B 0,C 180,E1 15238.585,E2 15238.585} C_VEL
LIN {X 0,Y 293.336,Z 790.13,A -85,B 0,C 180,E1 15244.667,E2 15244.667} C_VEL
LIN {X 0,Y 295.912,Z 782.477,A -85,B 0,C 180,E1 15251.521,E2 15251.521} C_VEL
LIN {X 0,Y 301.196,Z 768.762,A -85,B 0,C 180,E1 15258.718,E2 15258.718} C_VEL
LIN {X 0,Y 309.203,Z 749.337,A -85,B 0,C 180,E1 15265.324,E2 15265.324} C_VEL
LIN {X 0,Y 318.797,Z 726.152,A -85,B 0,C 180,E1 15270.757,E2 15270.757} C_VEL
LIN {X 0,Y 329.154,Z 698.824,A -85,B 0,C 180,E1 15275.288,E2 15275.288} C_VEL
LIN {X 0,Y 339.466,Z 667.155,A -85,B 0,C 180,E1 15278.982,E2 15278.982} C_VEL
LIN {X 0,Y 343.306,Z 651.508,A -85,B 0,C 180,E1 15280.445,E2 15280.445} C_VEL
LIN {X 0,Y 337.149,Z 625.935,A -85,B 0,C 180,E1 15285.112,E2 15285.112} C_VEL
LIN {X 0,Y 327.836,Z 602.754,A -85,B 0,C 180,E1 15290.463,E2 15290.463} C_VEL
LIN {X 0,Y 318.683,Z 585.75,A -85,B 0,C 180,E1 15296.036,E2 15296.036} C_VEL
LIN {X 0,Y 313.996,Z 578.702,A -85,B 0,C 180,E1 15299.599,E2 15299.599} C_VEL
LIN {X 0,Y 310.48,Z 572.606,A -85,B 0,C 180,E1 15303.535,E2 15303.535} C_VEL
LIN {X 0,Y 308.188,Z 571.799,A -85,B 0,C 180,E1 15312.64,E2 15312.64} C_VEL
LIN {X 0,Y 310.23,Z 573.64,A -85,B 0,C 180,E1 15316.443,E2 15316.443} C_VEL
LIN {X 0,Y 314.473,Z 579.741,A -85,B 0,C 180,E1 15320.815,E2 15320.815} C_VEL
LIN {X 0,Y 322.976,Z 593.042,A -85,B 0,C 180,E1 15326.367,E2 15326.367} C_VEL
LIN {X 0,Y 334.08,Z 612.887,A -85,B 0,C 180,E1 15331.835,E2 15331.835} C_VEL
LIN {X 0,Y 344.085,Z 636.896,A -85,B 0,C 180,E1 15336.428,E2 15336.428} C_VEL
LIN {X 0,Y 349.571,Z 656.778,A -85,B 0,C 180,E1 15339.462,E2 15339.462} C_VEL
LIN {X 0,Y 340.394,Z 692.816,A -85,B 0,C 180,E1 15342.054,E2 15342.054} C_VEL
LIN {X 0,Y 329.2,Z 728.046,A -85,B 0,C 180,E1 15345.752,E2 15345.752} C_VEL
LIN {X 0,Y 317.76,Z 759.903,A -85,B 0,C 180,E1 15350.57,E2 15350.57} C_VEL
LIN {X 0,Y 307.819,Z 786.537,A -85,B 0,C 180,E1 15356.22,E2 15356.22} C_VEL
LIN {X 0,Y 299.678,Z 809.564,A -85,B 0,C 180,E1 15363.054,E2 15363.054} C_VEL
LIN {X 0,Y 294.794,Z 826.359,A -85,B 0,C 180,E1 15370.13,E2 15370.13} C_VEL
LIN {X 0,Y 292.848,Z 836.882,A -85,B 0,C 180,E1 15376.595,E2 15376.595} C_VEL
LIN {X 0,Y 292.288,Z 842.941,A -85,B 0,C 180,E1 15382.586,E2 15382.586} C_VEL
LIN {X 0,Y 292.622,Z 845.739,A -85,B 0,C 180,E1 15390.002,E2 15390.002} C_VEL
LIN {X 0,Y 292.284,Z 843.078,A -85,B 0,C 180,E1 15397.418,E2 15397.418} C_VEL
LIN {X 0,Y 293.173,Z 834.961,A -85,B 0,C 180,E1 15404.916,E2 15404.916} C_VEL
LIN {X 0,Y 296.175,Z 821.085,A -85,B 0,C 180,E1 15412.439,E2 15412.439} C_VEL
LIN {X 0,Y 302.174,Z 801.769,A -85,B 0,C 180,E1 15419.489,E2 15419.489} C_VEL
LIN {X 0,Y 311.061,Z 776.673,A -85,B 0,C 180,E1 15425.91,E2 15425.91} C_VEL
LIN {X 0,Y 321.147,Z 748.111,A -85,B 0,C 180,E1 15431.138,E2 15431.138} C_VEL
LIN {X 0,Y 331.712,Z 715.951,A -85,B 0,C 180,E1 15435.316,E2 15435.316} C_VEL
LIN {X 0,Y 341.412,Z 680.895,A -85,B 0,C 180,E1 15438.515,E2 15438.515} C_VEL
LIN {X 0,Y 346.894,Z 655.607,A -85,B 0,C 180,E1 15440.2,E2 15440.2} C_VEL
LIN {X 0,Y 344.711,Z 648.523,A -85,B 0,C 180,E1 15441.194,E2 15441.194} C_VEL
LIN {X 0,Y 333.091,Z 635.96,A -85,B 0,C 180,E1 15444.279,E2 15444.279} C_VEL
LIN {X 0,Y 332.745,Z 635.149,A -85,B 0,C 180,E1 15444.406,E2 15444.406} C_VEL
LIN {X 0,Y 318.973,Z 606.479,A -85,B 0,C 180,E1 15449.315,E2 15449.315} C_VEL
LIN {X 0,Y 303.023,Z 580.507,A -85,B 0,C 180,E1 15454.82,E2 15454.82} C_VEL
LIN {X 0,Y 290.55,Z 562.559,A -85,B 0,C 180,E1 15459.7,E2 15459.7} C_VEL
LIN {X 0,Y 285.923,Z 556.076,A -85,B 0,C 180,E1 15461.77,E2 15461.77} C_VEL
LIN {X 0,Y 282.671,Z 551.389,A -85,B 0,C 180,E1 15463.341,E2 15463.341} C_VEL
LIN {X 0,Y 282.477,Z 549.53,A -85,B 0,C 180,E1 15463.552,E2 15463.552} C_VEL
LIN {X 0,Y 283.071,Z 549.53,A -85,B 0,C 180,E1 15470.774,E2 15470.774} C_VEL
LIN {X 0,Y 283.711,Z 549.53,A -85,B 0,C 180,E1 15476.926,E2 15476.926} C_VEL
LIN {X 0,Y 283.661,Z 549.53,A -85,B 0,C 180,E1 15483.023,E2 15483.023} C_VEL
LIN {X 0,Y 282.935,Z 549.53,A -85,B 0,C 180,E1 15492.289,E2 15492.289} C_VEL
LIN {X 0,Y 282.482,Z 549.53,A -85,B 0,C 180,E1 15498.663,E2 15498.663} C_VEL
LIN {X 0,Y 282.055,Z 549.53,A -85,B 0,C 180,E1 15505.306,E2 15505.306} C_VEL
LIN {X 0,Y 281.828,Z 549.53,A -85,B 0,C 180,E1 15512.335,E2 15512.335} C_VEL
LIN {X 0,Y 281.518,Z 549.53,A -85,B 0,C 180,E1 15519.989,E2 15519.989} C_VEL
LIN {X 0,Y 281.498,Z 549.53,A -85,B 0,C 180,E1 15528.579,E2 15528.579} C_VEL
LIN {X 0,Y 281.655,Z 551.192,A -85,B 0,C 180,E1 15529.091,E2 15529.091} C_VEL
LIN {X 0,Y 284.992,Z 556.012,A -85,B 0,C 180,E1 15530.723,E2 15530.723} C_VEL
LIN {X 0,Y 287.205,Z 558.583,A -85,B 0,C 180,E1 15531.707,E2 15531.707} C_VEL
LIN {X 0,Y 301.081,Z 578.28,A -85,B 0,C 180,E1 15537.394,E2 15537.394} C_VEL
LIN {X 0,Y 314.339,Z 601.058,A -85,B 0,C 180,E1 15542.596,E2 15542.596} C_VEL
LIN {X 0,Y 325.637,Z 627.168,A -85,B 0,C 180,E1 15547.549,E2 15547.549} C_VEL
LIN {X 0,Y 332.25,Z 650.382,A -85,B 0,C 180,E1 15551.46,E2 15551.46} C_VEL
LIN {X 0,Y 323.065,Z 684.6,A -85,B 0,C 180,E1 15554.939,E2 15554.939} C_VEL
LIN {X 0,Y 313.119,Z 714.223,A -85,B 0,C 180,E1 15559.235,E2 15559.235} C_VEL
LIN {X 0,Y 303.448,Z 739.786,A -85,B 0,C 180,E1 15564.468,E2 15564.468} C_VEL
LIN {X 0,Y 295.005,Z 761.457,A -85,B 0,C 180,E1 15570.824,E2 15570.824} C_VEL
LIN {X 0,Y 289.199,Z 777.445,A -85,B 0,C 180,E1 15577.806,E2 15577.806} C_VEL
LIN {X 0,Y 285.9,Z 788.099,A -85,B 0,C 180,E1 15585.3,E2 15585.3} C_VEL
LIN {X 0,Y 284.248,Z 792.949,A -85,B 0,C 180,E1 15591.813,E2 15591.813} C_VEL
LIN {X 0,Y 284.069,Z 793.879,A -85,B 0,C 180,E1 15598.558,E2 15598.558} C_VEL
LIN {X 0,Y 285.713,Z 790.458,A -85,B 0,C 180,E1 15605.516,E2 15605.516} C_VEL
LIN {X 0,Y 288.978,Z 781.63,A -85,B 0,C 180,E1 15613.075,E2 15613.075} C_VEL
LIN {X 0,Y 294.753,Z 767.591,A -85,B 0,C 180,E1 15620.166,E2 15620.166} C_VEL
LIN {X 0,Y 303.156,Z 748.556,A -85,B 0,C 180,E1 15626.556,E2 15626.556} C_VEL
LIN {X 0,Y 313.873,Z 723.841,A -85,B 0,C 180,E1 15632.262,E2 15632.262} C_VEL
LIN {X 0,Y 325.386,Z 694.08,A -85,B 0,C 180,E1 15637.003,E2 15637.003} C_VEL
LIN {X 0,Y 336,Z 661.459,A -85,B 0,C 180,E1 15640.579,E2 15640.579} C_VEL
LIN {X 0,Y 337.702,Z 655.382,A -85,B 0,C 180,E1 15641.124,E2 15641.124} C_VEL
LIN {X 0,Y 332.62,Z 631.847,A -85,B 0,C 180,E1 15645.577,E2 15645.577} C_VEL
LIN {X 0,Y 324.179,Z 608.978,A -85,B 0,C 180,E1 15651.053,E2 15651.053} C_VEL
LIN {X 0,Y 316.043,Z 592.7,A -85,B 0,C 180,E1 15656.638,E2 15656.638} C_VEL
LIN {X 0,Y 312.05,Z 586.111,A -85,B 0,C 180,E1 15660.023,E2 15660.023} C_VEL
LIN {X 0,Y 308.997,Z 580.328,A -85,B 0,C 180,E1 15663.812,E2 15663.812} C_VEL
LIN {X 0,Y 307.101,Z 579.632,A -85,B 0,C 180,E1 15672.796,E2 15672.796} C_VEL
LIN {X 0,Y 308.845,Z 581.418,A -85,B 0,C 180,E1 15676.155,E2 15676.155} C_VEL
LIN {X 0,Y 313.706,Z 589.389,A -85,B 0,C 180,E1 15681.329,E2 15681.329} C_VEL
LIN {X 0,Y 320.407,Z 600.149,A -85,B 0,C 180,E1 15685.92,E2 15685.92} C_VEL
LIN {X 0,Y 330.856,Z 619.88,A -85,B 0,C 180,E1 15691.461,E2 15691.461} C_VEL
LIN {X 0,Y 339.731,Z 643.475,A -85,B 0,C 180,E1 15696.07,E2 15696.07} C_VEL
LIN {X 0,Y 343.894,Z 659.505,A -85,B 0,C 180,E1 15698.62,E2 15698.62} C_VEL
LIN {X 0,Y 333.733,Z 696.673,A -85,B 0,C 180,E1 15701.41,E2 15701.41} C_VEL
LIN {X 0,Y 321.87,Z 731.752,A -85,B 0,C 180,E1 15705.315,E2 15705.315} C_VEL
LIN {X 0,Y 310.733,Z 761.067,A -85,B 0,C 180,E1 15709.952,E2 15709.952} C_VEL
LIN {X 0,Y 300.333,Z 787.55,A -85,B 0,C 180,E1 15715.793,E2 15715.793} C_VEL
LIN {X 0,Y 292.023,Z 809.899,A -85,B 0,C 180,E1 15722.705,E2 15722.705} C_VEL
LIN {X 0,Y 286.943,Z 826.466,A -85,B 0,C 180,E1 15730.014,E2 15730.014} C_VEL
LIN {X 0,Y 285.033,Z 836.175,A -85,B 0,C 180,E1 15736.22,E2 15736.22} C_VEL
LIN {X 0,Y 284.416,Z 842.235,A -85,B 0,C 180,E1 15742.38,E2 15742.38} C_VEL
LIN {X 0,Y 284.751,Z 845.027,A -85,B 0,C 180,E1 15750.002,E2 15750.002} C_VEL
LIN {X 0,Y 284.41,Z 842.348,A -85,B 0,C 180,E1 15757.625,E2 15757.625} C_VEL
LIN {X 0,Y 285.368,Z 834.191,A -85,B 0,C 180,E1 15765.334,E2 15765.334} C_VEL
LIN {X 0,Y 288.56,Z 820.46,A -85,B 0,C 180,E1 15772.964,E2 15772.964} C_VEL
LIN {X 0,Y 294.993,Z 800.854,A -85,B 0,C 180,E1 15780.271,E2 15780.271} C_VEL
LIN {X 0,Y 303.946,Z 776.82,A -85,B 0,C 180,E1 15786.57,E2 15786.57} C_VEL
LIN {X 0,Y 314.615,Z 747.966,A -85,B 0,C 180,E1 15791.954,E2 15791.954} C_VEL
LIN {X 0,Y 325.476,Z 716.091,A -85,B 0,C 180,E1 15796.171,E2 15796.171} C_VEL
LIN {X 0,Y 335.63,Z 680.718,A -85,B 0,C 180,E1 15799.438,E2 15799.438} C_VEL
LIN {X 0,Y 340.716,Z 658.039,A -85,B 0,C 180,E1 15800.99,E2 15800.99} C_VEL
LIN {X 0,Y 332.745,Z 635.149,A -85,B 0,C 180,E1 15804.406,E2 15804.406} C_VEL
LIN {X 0,Y 327.374,Z 627.742,A -85,B 0,C 180,E1 15806.04,E2 15806.04} C_VEL
LIN {X 0,Y 318.106,Z 618.493,A -85,B 0,C 180,E1 15808.718,E2 15808.718} C_VEL
LIN {X 0,Y 317.353,Z 617.072,A -85,B 0,C 180,E1 15808.992,E2 15808.992} C_VEL
LIN {X 0,Y 301.29,Z 588.819,A -85,B 0,C 180,E1 15814.92,E2 15814.92} C_VEL
LIN {X 0,Y 287.559,Z 569.074,A -85,B 0,C 180,E1 15820.432,E2 15820.432} C_VEL
LIN {X 0,Y 282.648,Z 562.425,A -85,B 0,C 180,E1 15822.702,E2 15822.702} C_VEL
LIN {X 0,Y 278.62,Z 556.371,A -85,B 0,C 180,E1 15824.768,E2 15824.768} C_VEL
LIN {X 0,Y 275.08,Z 551.768,A -85,B 0,C 180,E1 15826.696,E2 15826.696} C_VEL
LIN {X 0,Y 274.804,Z 549.53,A -85,B 0,C 180,E1 15827.086,E2 15827.086} C_VEL
LIN {X 0,Y 275.394,Z 549.53,A -85,B 0,C 180,E1 15833.684,E2 15833.684} C_VEL
LIN {X 0,Y 275.979,Z 549.53,A -85,B 0,C 180,E1 15839.974,E2 15839.974} C_VEL
LIN {X 0,Y 275.451,Z 549.53,A -85,B 0,C 180,E1 15846.263,E2 15846.263} C_VEL
LIN {X 0,Y 274.973,Z 549.53,A -85,B 0,C 180,E1 15852.651,E2 15852.651} C_VEL
LIN {X 0,Y 274.329,Z 549.53,A -85,B 0,C 180,E1 15860.745,E2 15860.745} C_VEL
LIN {X 0,Y 273.946,Z 549.53,A -85,B 0,C 180,E1 15869.682,E2 15869.682} C_VEL
LIN {X 0,Y 273.633,Z 549.53,A -85,B 0,C 180,E1 15877.302,E2 15877.302} C_VEL
LIN {X 0,Y 273.564,Z 549.577,A -85,B 0,C 180,E1 15885.338,E2 15885.338} C_VEL
LIN {X 0,Y 275.551,Z 554.825,A -85,B 0,C 180,E1 15886.653,E2 15886.653} C_VEL
LIN {X 0,Y 279,Z 558.252,A -85,B 0,C 180,E1 15888.422,E2 15888.422} C_VEL
LIN {X 0,Y 285.658,Z 567.488,A -85,B 0,C 180,E1 15891.641,E2 15891.641} C_VEL
LIN {X 0,Y 297.407,Z 584.321,A -85,B 0,C 180,E1 15896.725,E2 15896.725} C_VEL
LIN {X 0,Y 310.71,Z 608.316,A -85,B 0,C 180,E1 15902.361,E2 15902.361} C_VEL
LIN {X 0,Y 320.991,Z 634.034,A -85,B 0,C 180,E1 15907.345,E2 15907.345} C_VEL
LIN {X 0,Y 325.989,Z 654.451,A -85,B 0,C 180,E1 15910.85,E2 15910.85} C_VEL
LIN {X 0,Y 315.991,Z 688.3,A -85,B 0,C 180,E1 15914.416,E2 15914.416} C_VEL
LIN {X 0,Y 305.481,Z 718.13,A -85,B 0,C 180,E1 15918.962,E2 15918.962} C_VEL
LIN {X 0,Y 294.94,Z 744.606,A -85,B 0,C 180,E1 15924.757,E2 15924.757} C_VEL
LIN {X 0,Y 286.593,Z 765.034,A -85,B 0,C 180,E1 15931.302,E2 15931.302} C_VEL
LIN {X 0,Y 280.785,Z 780.381,A -85,B 0,C 180,E1 15938.658,E2 15938.658} C_VEL
LIN {X 0,Y 277.905,Z 789.507,A -85,B 0,C 180,E1 15945.751,E2 15945.751} C_VEL
LIN {X 0,Y 276.251,Z 793.924,A -85,B 0,C 180,E1 15952.478,E2 15952.478} C_VEL
LIN {X 0,Y 276.29,Z 794.399,A -85,B 0,C 180,E1 15959.44,E2 15959.44} C_VEL
LIN {X 0,Y 278.193,Z 790.525,A -85,B 0,C 180,E1 15966.629,E2 15966.629} C_VEL
LIN {X 0,Y 281.79,Z 781.566,A -85,B 0,C 180,E1 15974.117,E2 15974.117} C_VEL
LIN {X 0,Y 287.776,Z 767.948,A -85,B 0,C 180,E1 15981.049,E2 15981.049} C_VEL
LIN {X 0,Y 296.687,Z 749.003,A -85,B 0,C 180,E1 15987.497,E2 15987.497} C_VEL
LIN {X 0,Y 307.906,Z 724.369,A -85,B 0,C 180,E1 15993.26,E2 15993.26} C_VEL
LIN {X 0,Y 319.751,Z 695.083,A -85,B 0,C 180,E1 15997.977,E2 15997.977} C_VEL
LIN {X 0,Y 330.555,Z 663.32,A -85,B 0,C 180,E1 16001.511,E2 16001.511} C_VEL
LIN {X 0,Y 331.929,Z 657.71,A -85,B 0,C 180,E1 16002.1,E2 16002.1} C_VEL
LIN {X 0,Y 327.262,Z 634.779,A -85,B 0,C 180,E1 16006.696,E2 16006.696} C_VEL
LIN {X 0,Y 319.87,Z 613.81,A -85,B 0,C 180,E1 16012.09,E2 16012.09} C_VEL
LIN {X 0,Y 313.239,Z 599.441,A -85,B 0,C 180,E1 16017.262,E2 16017.262} C_VEL
LIN {X 0,Y 309.787,Z 593.208,A -85,B 0,C 180,E1 16020.629,E2 16020.629} C_VEL
LIN {X 0,Y 307.228,Z 588.024,A -85,B 0,C 180,E1 16024.307,E2 16024.307} C_VEL
LIN {X 0,Y 305.889,Z 587.455,A -85,B 0,C 180,E1 16032.847,E2 16032.847} C_VEL
LIN {X 0,Y 307.438,Z 589.28,A -85,B 0,C 180,E1 16035.956,E2 16035.956} C_VEL
LIN {X 0,Y 311.765,Z 597.016,A -85,B 0,C 180,E1 16041.04,E2 16041.04} C_VEL
LIN {X 0,Y 318,Z 607.763,A -85,B 0,C 180,E1 16045.634,E2 16045.634} C_VEL
LIN {X 0,Y 327.155,Z 626.385,A -85,B 0,C 180,E1 16050.987,E2 16050.987} C_VEL
LIN {X 0,Y 335.428,Z 650.522,A -85,B 0,C 180,E1 16055.808,E2 16055.808} C_VEL
LIN {X 0,Y 338.064,Z 662.568,A -85,B 0,C 180,E1 16057.767,E2 16057.767} C_VEL
LIN {X 0,Y 327.588,Z 698.827,A -85,B 0,C 180,E1 16060.603,E2 16060.603} C_VEL
LIN {X 0,Y 315.679,Z 732.377,A -85,B 0,C 180,E1 16064.438,E2 16064.438} C_VEL
LIN {X 0,Y 303.661,Z 762.516,A -85,B 0,C 180,E1 16069.355,E2 16069.355} C_VEL
LIN {X 0,Y 292.683,Z 789,A -85,B 0,C 180,E1 16075.452,E2 16075.452} C_VEL
LIN {X 0,Y 283.963,Z 811.27,A -85,B 0,C 180,E1 16082.722,E2 16082.722} C_VEL
LIN {X 0,Y 278.543,Z 828.575,A -85,B 0,C 180,E1 16091.034,E2 16091.034} C_VEL
LIN {X 0,Y 276.769,Z 838.965,A -85,B 0,C 180,E1 16099,E2 16099} C_VEL
LIN {X 0,Y 276.539,Z 843.852,A -85,B 0,C 180,E1 16106.874,E2 16106.874} C_VEL
LIN {X 0,Y 276.897,Z 844.317,A -85,B 0,C 180,E1 16110.002,E2 16110.002} C_VEL
LIN {X 0,Y 276.529,Z 841.615,A -85,B 0,C 180,E1 16117.843,E2 16117.843} C_VEL
LIN {X 0,Y 277.573,Z 833.417,A -85,B 0,C 180,E1 16125.775,E2 16125.775} C_VEL
LIN {X 0,Y 281.149,Z 819.295,A -85,B 0,C 180,E1 16133.761,E2 16133.761} C_VEL
LIN {X 0,Y 287.961,Z 799.767,A -85,B 0,C 180,E1 16141.143,E2 16141.143} C_VEL
LIN {X 0,Y 297.32,Z 775.724,A -85,B 0,C 180,E1 16147.523,E2 16147.523} C_VEL
LIN {X 0,Y 308.268,Z 747.361,A -85,B 0,C 180,E1 16152.883,E2 16152.883} C_VEL
LIN {X 0,Y 319.639,Z 715.251,A -85,B 0,C 180,E1 16157.159,E2 16157.159} C_VEL
LIN {X 0,Y 329.869,Z 680.652,A -85,B 0,C 180,E1 16160.379,E2 16160.379} C_VEL
LIN {X 0,Y 334.564,Z 660.842,A -85,B 0,C 180,E1 16161.775,E2 16161.775} C_VEL
LIN {X 0,Y 323.894,Z 631.096,A -85,B 0,C 180,E1 16166.492,E2 16166.492} C_VEL
LIN {X 0,Y 317.353,Z 617.072,A -85,B 0,C 180,E1 16168.992,E2 16168.992} C_VEL
LIN {X 0,Y 313.252,Z 613.411,A -85,B 0,C 180,E1 16170.244,E2 16170.244} C_VEL
LIN {X 0,Y 306.303,Z 609.665,A -85,B 0,C 180,E1 16172.273,E2 16172.273} C_VEL
LIN {X 0,Y 305.742,Z 608.81,A -85,B 0,C 180,E1 16172.476,E2 16172.476} C_VEL
LIN {X 0,Y 291.978,Z 586.196,A -85,B 0,C 180,E1 16177.973,E2 16177.973} C_VEL
LIN {X 0,Y 280.453,Z 569.67,A -85,B 0,C 180,E1 16183.167,E2 16183.167} C_VEL
LIN {X 0,Y 275.761,Z 563.176,A -85,B 0,C 180,E1 16185.62,E2 16185.62} C_VEL
LIN {X 0,Y 272.274,Z 557.48,A -85,B 0,C 180,E1 16187.676,E2 16187.676} C_VEL
LIN {X 0,Y 267.738,Z 552.355,A -85,B 0,C 180,E1 16190.49,E2 16190.49} C_VEL
LIN {X 0,Y 267.265,Z 549.53,A -85,B 0,C 180,E1 16191.216,E2 16191.216} C_VEL
LIN {X 0,Y 267.847,Z 549.53,A -85,B 0,C 180,E1 16196.744,E2 16196.744} C_VEL
LIN {X 0,Y 267.809,Z 549.53,A -85,B 0,C 180,E1 16203.202,E2 16203.202} C_VEL
LIN {X 0,Y 267.242,Z 549.53,A -85,B 0,C 180,E1 16209.723,E2 16209.723} C_VEL
LIN {X 0,Y 266.763,Z 549.53,A -85,B 0,C 180,E1 16216.398,E2 16216.398} C_VEL
LIN {X 0,Y 266.099,Z 549.53,A -85,B 0,C 180,E1 16224.854,E2 16224.854} C_VEL
LIN {X 0,Y 265.812,Z 549.53,A -85,B 0,C 180,E1 16231.615,E2 16231.615} C_VEL
LIN {X 0,Y 265.663,Z 549.53,A -85,B 0,C 180,E1 16238.623,E2 16238.623} C_VEL
LIN {X 0,Y 265.715,Z 550.117,A -85,B 0,C 180,E1 16241.116,E2 16241.116} C_VEL
LIN {X 0,Y 267.938,Z 555.123,A -85,B 0,C 180,E1 16242.811,E2 16242.811} C_VEL
LIN {X 0,Y 271.271,Z 558.058,A -85,B 0,C 180,E1 16244.817,E2 16244.817} C_VEL
LIN {X 0,Y 275.184,Z 563.614,A -85,B 0,C 180,E1 16247.085,E2 16247.085} C_VEL
LIN {X 0,Y 283.43,Z 575.029,A -85,B 0,C 180,E1 16251.308,E2 16251.308} C_VEL
LIN {X 0,Y 295.223,Z 593.073,A -85,B 0,C 180,E1 16256.751,E2 16256.751} C_VEL
LIN {X 0,Y 306.922,Z 615.873,A -85,B 0,C 180,E1 16262.174,E2 16262.174} C_VEL
LIN {X 0,Y 316.28,Z 641.413,A -85,B 0,C 180,E1 16267.26,E2 16267.26} C_VEL
LIN {X 0,Y 319.704,Z 657.395,A -85,B 0,C 180,E1 16270.088,E2 16270.088} C_VEL
LIN {X 0,Y 309.377,Z 690.76,A -85,B 0,C 180,E1 16273.71,E2 16273.71} C_VEL
LIN {X 0,Y 298.546,Z 720.16,A -85,B 0,C 180,E1 16278.333,E2 16278.333} C_VEL
LIN {X 0,Y 288.075,Z 745.281,A -85,B 0,C 180,E1 16283.984,E2 16283.984} C_VEL
LIN {X 0,Y 279.311,Z 765.718,A -85,B 0,C 180,E1 16290.667,E2 16290.667} C_VEL
LIN {X 0,Y 273.093,Z 781.27,A -85,B 0,C 180,E1 16298.325,E2 16298.325} C_VEL
LIN {X 0,Y 269.906,Z 790.901,A -85,B 0,C 180,E1 16306.23,E2 16306.23} C_VEL
LIN {X 0,Y 268.278,Z 794.9,A -85,B 0,C 180,E1 16313.185,E2 16313.185} C_VEL
LIN {X 0,Y 268.553,Z 794.911,A -85,B 0,C 180,E1 16320.376,E2 16320.376} C_VEL
LIN {X 0,Y 270.78,Z 790.546,A -85,B 0,C 180,E1 16327.805,E2 16327.805} C_VEL
LIN {X 0,Y 274.876,Z 781.02,A -85,B 0,C 180,E1 16335.531,E2 16335.531} C_VEL
LIN {X 0,Y 282.487,Z 765.226,A -85,B 0,C 180,E1 16343.249,E2 16343.249} C_VEL
LIN {X 0,Y 292.788,Z 744.359,A -85,B 0,C 180,E1 16349.886,E2 16349.886} C_VEL
LIN {X 0,Y 304.897,Z 718.495,A -85,B 0,C 180,E1 16355.489,E2 16355.489} C_VEL
LIN {X 0,Y 317.28,Z 688.274,A -85,B 0,C 180,E1 16359.996,E2 16359.996} C_VEL
LIN {X 0,Y 326.254,Z 660.755,A -85,B 0,C 180,E1 16362.986,E2 16362.986} C_VEL
LIN {X 0,Y 322.161,Z 638.235,A -85,B 0,C 180,E1 16367.76,E2 16367.76} C_VEL
LIN {X 0,Y 315.333,Z 617.342,A -85,B 0,C 180,E1 16373.498,E2 16373.498} C_VEL
LIN {X 0,Y 309.895,Z 605.337,A -85,B 0,C 180,E1 16378.367,E2 16378.367} C_VEL
LIN {X 0,Y 307.462,Z 600.392,A -85,B 0,C 180,E1 16381.147,E2 16381.147} C_VEL
LIN {X 0,Y 305.313,Z 595.581,A -85,B 0,C 180,E1 16384.835,E2 16384.835} C_VEL
LIN {X 0,Y 304.675,Z 595.393,A -85,B 0,C 180,E1 16393.628,E2 16393.628} C_VEL
LIN {X 0,Y 305.756,Z 597.253,A -85,B 0,C 180,E1 16395.879,E2 16395.879} C_VEL
LIN {X 0,Y 309.693,Z 604.491,A -85,B 0,C 180,E1 16400.72,E2 16400.72} C_VEL
LIN {X 0,Y 315.377,Z 615.224,A -85,B 0,C 180,E1 16405.337,E2 16405.337} C_VEL
LIN {X 0,Y 323.434,Z 632.855,A -85,B 0,C 180,E1 16410.508,E2 16410.508} C_VEL
LIN {X 0,Y 331.054,Z 657.572,A -85,B 0,C 180,E1 16415.57,E2 16415.57} C_VEL
LIN {X 0,Y 332.328,Z 665.613,A -85,B 0,C 180,E1 16416.888,E2 16416.888} C_VEL
LIN {X 0,Y 321.5,Z 701.116,A -85,B 0,C 180,E1 16419.773,E2 16419.773} C_VEL
LIN {X 0,Y 308.664,Z 735.412,A -85,B 0,C 180,E1 16423.857,E2 16423.857} C_VEL
LIN {X 0,Y 295.568,Z 766.379,A -85,B 0,C 180,E1 16429.206,E2 16429.206} C_VEL
